# B&R Automation Studio project BR_ZBM1
Automation Studio 4.1.5.68 SP

## Configuration Config1

CPU , AutomationRuntime K4.06, Build 4.1.2

### Task classes (Cpu.sw)
```
Cyclic#4 (cycle 100000 us, tolerance 100000 us):
  BU_2 <- BunchUnits.BU_2.prg
  can_diag <- Exceptionhandling.can_diag.prg
  SC_2 <- BunchUnits.SC_2.prg
VcDataObjects: Mobile <- Visualisation.Mobile.dob
Binaries: asfw, ashwd, arconfig, sysconf, iomap
Libraries: standard, astime, runtime, asieccon, Hardware
```

### Hardware
```
X20CP1586 : X20CP1586 v1.0.5.0
  Connector IF2:
    ActivateDevice = 1
    Mode = Manual
    InternetAddress = 192.168.0.1
    SubnetMask = 255.255.255.0
  Cyclic1Duration = 1000
  Cyclic1Tolerance = 10000
  Cyclic2Duration = 20000
  Cyclic2Tolerance = 20000
  Cyclic3Duration = 50000
  Cyclic3Tolerance = 50000
  Cyclic4Duration = 100000
  Cyclic4Tolerance = 100000
  Cyclic5Duration = 200000
  Cyclic5Tolerance = 200000
  Cyclic6Duration = 500000
  Cyclic6Tolerance = 500000
  Cyclic7Duration = 1000000
  Cyclic7Tolerance = 1000000
  Cyclic8Duration = 10000
  Cyclic8Tolerance = 30000000
```

### IoMap.iom - X20CP1586/IoMap.iom
```iecst
(********************************************************************
 * COPYRIGHT -- Bernecker + Rainer
 ********************************************************************
 * File: IoMap.iom
 * Author: frankenj
 * Created: December 04, 2014
 ********************************************************************
 * IO mapping file
 ********************************************************************)
VAR_CONFIG
	::myPulseUse:linkedSystemTime AT %ID."X20CP1586".SystemTime;
END_VAR
```

## Configuration X20

CPU X20CP1585, AutomationRuntime C4.09, Build 4.1.2

### Task classes (Cpu.sw)
```
Cyclic#1 (cycle 1000 us, tolerance 0 us):
  Shiftregis <- MainControlUnit.Shiftregister.prg  // Control for chain sensor
  Simulation <- MainControlUnit.Simulation.prg
  Main <- MainControlUnit.Main.prg
Cyclic#2 (cycle 5000 us, tolerance 0 us):
  IOpolling <- IOHandling.IOpolling.prg
  BeltContro <- MainBeltUnit.BeltControl.prg
Cyclic#3 (cycle 50000 us, tolerance 0 us):
  RS_I <- BunchUnits.RS_I.prg
  BU_1 <- BunchUnits.BU_1.prg
  SC_1 <- BunchUnits.SC_1.prg
  BU_2 <- BunchUnits.BU_2.prg
  SC_2 <- BunchUnits.SC_2.prg
  BU_3 <- BunchUnits.BU_3.prg
  SC_3 <- BunchUnits.SC_3.prg
  BU_4 <- BunchUnits.BU_4.prg
  SC_4 <- BunchUnits.SC_4.prg
  BU_5 <- BunchUnits.BU_5.prg
  SC_5 <- BunchUnits.SC_5.prg
  BU_6 <- BunchUnits.BU_6.prg
  SC_6 <- BunchUnits.SC_6.prg
  BU_7 <- BunchUnits.BU_7.prg
  SC_7 <- BunchUnits.SC_7.prg
  BU_8 <- BunchUnits.BU_8.prg
  SC_8 <- BunchUnits.SC_8.prg
  BU_9 <- BunchUnits.BU_9.prg
  SC_9 <- BunchUnits.SC_9.prg
  BU_10 <- BunchUnits.BU_10.prg
  SC_10 <- BunchUnits.SC_10.prg
Cyclic#4 (cycle 100000 us, tolerance 0 us):
  ErrorHandl <- Exceptionhandling.ErrorHandling.prg
  can_diag <- Exceptionhandling.can_diag.prg
Cyclic#5 (cycle 10000 us, tolerance 30000000 us):
  Init <- BunchUnits.Init.prg
  Sender <- Lichtkrant.Sender.prg
VcDataObjects: BU_Gui <- Visualisation.BU_Gui_Resized.dob [disabled], Mobile <- Visualisation.Mobile.dob [disabled]
Binaries: OpcUaMap, sysconf, iomap, ashwd, asfw, arconfig, asnxdb2, vcchspot, asnxdb1, vccbar, vcclbox, vcchtml, vccstr, vccline, vccscale, vccalarm, vccgauge, vccurl, vcxml, vcpfar00, vccnum, arialbd, vcdsloc, vcfntttf, vcdsint, vcshared, vcrt, vcbclass, vcfile, vccbtn, vcresman, vcalarm, vcpdsw, arial, vccovl, vcgclass, Mobile02, Mobile03, vccddbox, vccpopup, vccdt, vcctext, vccshape, vccbmp, vcctrend, BU_Gui02, BU_Gui03, vccslider, vcmgr, vcnet, vcpkat, vctcal, BU_Gui01, vcpdvnc, vcpfx20, Mobile01
Libraries: sys_lib, Runtime, astime, asieccon, AsTCP, brsystem, asstring, standard, PulsGen, AsNxCoM, Inverter, BULib, Servo, SDO, dvframe, Lichtkrant, Chain, AsBrStr, hex2dec, Serial, SensContr, MBU_lib, IecCheck, AsArLog, Hardware, dataobj, fileio, ashw
```

### Hardware
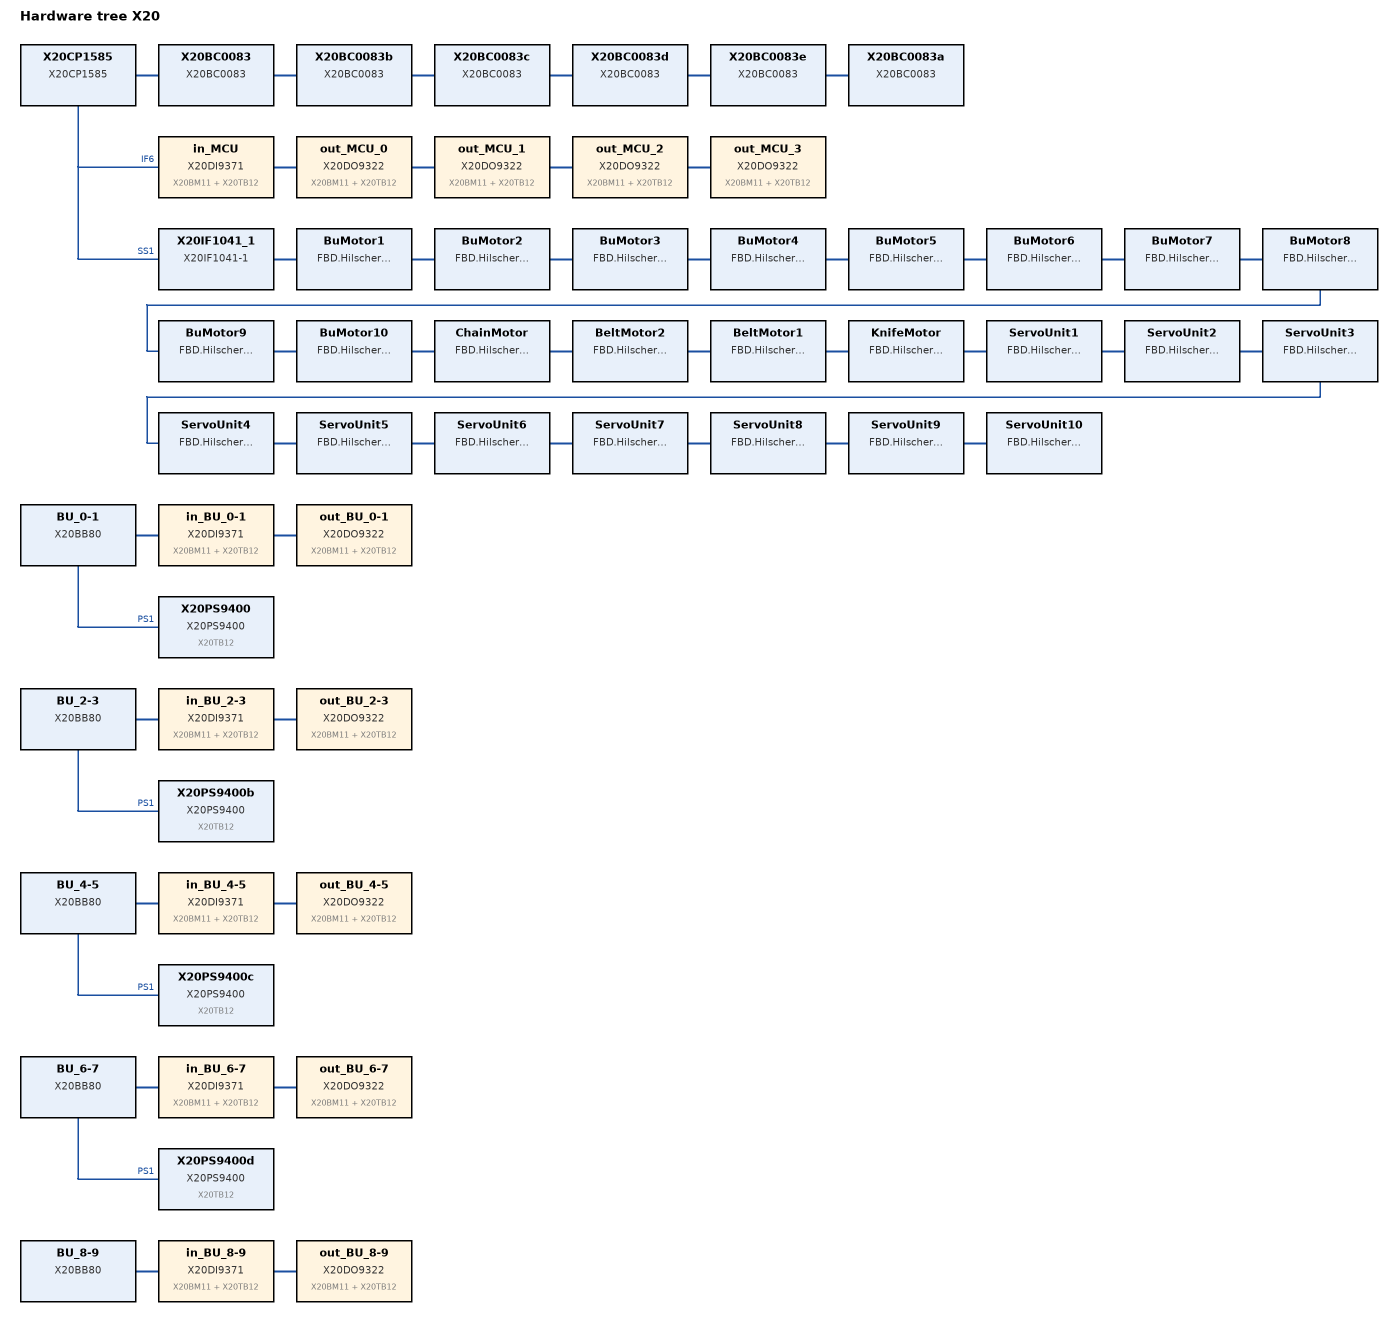
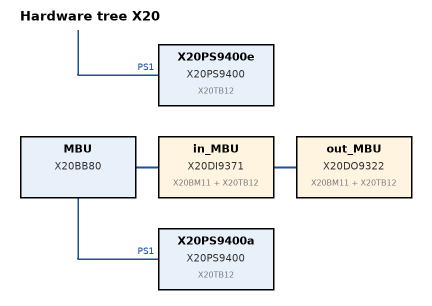
```
BeltMotor1 : FBD.Hilscher.COGenSlaveDTM.ACOPOSinverter X64 (ACOPOSinverter_X64.eds) v0.0.0.0 (OrderNumber=ACOPOSinverter_X64__ACOPOSinverter_X64_eds_)  [CAN1 -> BeltMotor2.CAN2 (NodeNumber=4)]
  DtmId = 0e41fe58-9b29-4e80-aa17-b3b9a602be41
  ChannelBlocks_54c748ae-a862-45bf-bd05-307df38cf45a  // Receive PDO1 parameter
  IO_aca35ca7-9daa-4f2c-a263-cb1312a79025  // 2 Byte(s)
  ChannelBlocks_6fc9c6dd-ef6a-4241-a49b-47093041261e  // Receive PDO6 parameter
  IO_a09422e8-9296-4dde-995f-c21dba077c83  // 2 Byte(s)
  IO_c6b60006-1097-4b2b-99a2-873ae92355e9  // 2 Byte(s)
  IO_be17ac07-0c86-4ed7-8a83-77242752eabc  // 2 Byte(s)
  ChannelBlocks_0de3404d-a2ba-475d-9759-ce1c75ca456f  // Transmit PDO1 parameter
  IO_d4d6ac5b-6312-46c0-bea3-1feb3fe2ff1b  // 2 Byte(s)
  ChannelBlocks_35f5ad43-0655-49b5-a722-94d15f201f4c  // Transmit PDO6 parameter
  IO_54646803-abb9-4e9d-b295-57a01534b6c3  // 2 Byte(s)
  IO_ae920d2b-a2b1-4de3-a1c4-e574386f93fb  // 2 Byte(s)
  IO_47f71d08-67d5-4a29-b608-1e0426a373c3  // 2 Byte(s)
  IO_76edcae2-a5b3-42ff-aea4-90ff8a7df386  // 2 Byte(s)
BeltMotor2 : FBD.Hilscher.COGenSlaveDTM.ACOPOSinverter X64 (ACOPOSinverter_X64.eds) v0.0.0.0 (OrderNumber=ACOPOSinverter_X64__ACOPOSinverter_X64_eds_)  [CAN1 -> ChainMotor.CAN2 (NodeNumber=5)]
  DtmId = 5224c894-1ef8-4fa5-9f2e-7023e8237f50
  ChannelBlocks_54ef21bf-51ac-4b79-9d7d-aaf36440fde1  // Receive PDO1 parameter
  IO_08901fce-ce4a-45a7-8fa1-4352fddaeca0  // 2 Byte(s)
  ChannelBlocks_5fdfdc2d-6504-40c7-b6e9-5c26043bbabb  // Receive PDO6 parameter
  IO_7efb87b6-7525-4814-82a4-a00de786267e  // 2 Byte(s)
  IO_1c5a6fdf-985c-41b4-867c-db4a3086964a  // 2 Byte(s)
  IO_89f973fb-223e-4f5d-b0cf-d7557db3c308  // 2 Byte(s)
  ChannelBlocks_ff6de664-0730-4c0c-a004-c59824083d59  // Transmit PDO1 parameter
  IO_6a6c6cea-e364-4156-9bd8-734b31d4d8b2  // 2 Byte(s)
  ChannelBlocks_b2f2cbd0-76eb-4694-9316-88ecd34e890c  // Transmit PDO6 parameter
  IO_27630f78-04b9-4817-a004-ac8ed4a34943  // 2 Byte(s)
  IO_a532a8b0-ae79-4199-8f10-aceb97e86d8c  // 2 Byte(s)
  IO_80c1adba-b4c6-4671-a8d4-c5debac3ab04  // 2 Byte(s)
  IO_db551fcc-40d8-4d75-964b-d0c34238111c  // 2 Byte(s)
BU_0-1 : X20BB80 v1.0.0.2
  Connector IF1:
    BusLength = 100
BU_2-3 : X20BB80 v1.0.0.2
BU_4-5 : X20BB80 v1.0.0.2
BU_6-7 : X20BB80 v1.0.0.2
BU_8-9 : X20BB80 v1.0.0.2
BuMotor1 : FBD.Hilscher.COGenSlaveDTM.ACOPOSinverter X64 (ACOPOSinverter_X64.eds) v0.0.0.0 (OrderNumber=ACOPOSinverter_X64__ACOPOSinverter_X64_eds_)  [CAN1 -> X20IF1041_1.IF1 (NodeNumber=10)]
  DtmId = 41eacdba-3555-4f40-ac61-2c8428ea58b2
  ChannelBlocks_b9ddc844-9481-4af5-a747-25b3e2109658  // Receive PDO1 parameter
  IO_7b4bc88c-5ce5-4aaa-a58d-90f33b48a65c  // 2 Byte(s)
  ChannelBlocks_8b5f3c6e-1732-4951-a210-c4de25588974  // Receive PDO6 parameter
  IO_39a2cd53-b850-4b06-8776-b6d11eb43720  // 2 Byte(s)
  IO_30629477-0436-4440-ba53-af916bfbef45  // 2 Byte(s)
  IO_eda63b9e-3d56-4a36-8c45-b6b1969d639a  // 2 Byte(s)
  ChannelBlocks_f1365d26-9917-401f-a453-e6262fccb88e  // Transmit PDO1 parameter
  IO_8b996910-5de3-45a7-9e18-c98469aeffd6  // 2 Byte(s)
  ChannelBlocks_48485091-4447-4b08-b8f7-2a8039d8dcd2  // Transmit PDO6 parameter
  IO_be2a3e1f-8d08-4dea-a2d2-a29b4de4c830  // 2 Byte(s)
  IO_55fef0e3-e778-4333-8784-725b71533f49  // 2 Byte(s)
  IO_626eea93-30a0-479c-9321-2dd4622e8684  // 2 Byte(s)
  IO_53a93a48-f76d-4478-8b66-bfaf7ee8cb03  // 2 Byte(s)
BuMotor10 : FBD.Hilscher.COGenSlaveDTM.ACOPOSinverter X64 (ACOPOSinverter_X64.eds) v0.0.0.0 (OrderNumber=ACOPOSinverter_X64__ACOPOSinverter_X64_eds_)  [CAN1 -> BuMotor9.CAN2 (NodeNumber=28)]
  DtmId = 334ec416-5c16-4925-9ab1-88c2f19d51fb
  ChannelBlocks_ac9c813b-77a1-48ff-9722-79a7e36309a3  // Receive PDO1 parameter
  IO_4aa75d45-937a-4143-8e5e-5239ec3df5d5  // 2 Byte(s)
  ChannelBlocks_bd99a9ef-60c2-4465-b2ca-5589d312d023  // Receive PDO6 parameter
  IO_10874e3a-ea7a-435e-b16d-3cfd83cd96d2  // 2 Byte(s)
  IO_a0da98ff-73a6-482d-a789-9eea3a9ef5ec  // 2 Byte(s)
  IO_a035e9e4-fedc-44f8-8d04-fa4482e8e6f6  // 2 Byte(s)
  ChannelBlocks_c4ede1fb-b8c3-46bc-aa40-d6c07d995dd8  // Transmit PDO1 parameter
  IO_3a67936d-7775-49f5-8896-9a8e4e400f8a  // 2 Byte(s)
  ChannelBlocks_4cda3d3d-ce84-47df-a9c8-383005e5aed1  // Transmit PDO6 parameter
  IO_f52c2df5-83ca-4265-9fb6-a04d781d80b2  // 2 Byte(s)
  IO_496498d8-ae6d-4630-839d-faafd4532c16  // 2 Byte(s)
  IO_a3e387be-6efa-4130-b18c-b95da0514b42  // 2 Byte(s)
  IO_b0e32a9b-b548-480f-ab2f-b0d362bbdba9  // 2 Byte(s)
BuMotor2 : FBD.Hilscher.COGenSlaveDTM.ACOPOSinverter X64 (ACOPOSinverter_X64.eds) v0.0.0.0 (OrderNumber=ACOPOSinverter_X64__ACOPOSinverter_X64_eds_)  [CAN1 -> BuMotor1.CAN2 (NodeNumber=12)]
  DtmId = e1ce438d-8ff1-4ad6-81a8-1a105d1b79ee
  ChannelBlocks_303446a4-05f8-4f0b-b2b4-7c1333c2b877  // Receive PDO1 parameter
  IO_edbfdedc-cf52-4617-8a63-87053fac3909  // 2 Byte(s)
  ChannelBlocks_72fe8bc7-9e89-4c3c-9af8-bb7ce4d6a99e  // Receive PDO6 parameter
  IO_7fc3c5cf-f8f6-4322-9a74-de616acc70eb  // 2 Byte(s)
  IO_f67c0509-47e2-4490-9eac-614590cde9d6  // 2 Byte(s)
  IO_987d5f71-5d59-414d-b133-eb996a41fb68  // 2 Byte(s)
  ChannelBlocks_1b47f333-0257-4114-959e-33d260186bf4  // Transmit PDO1 parameter
  IO_6f79accf-2d80-4323-98c0-77cea77bfb60  // 2 Byte(s)
  ChannelBlocks_efe37a9e-d3f3-48e1-a345-23b1c1da338c  // Transmit PDO6 parameter
  IO_a5a00cb8-1081-40a9-aa27-5251b345f7d4  // 2 Byte(s)
  IO_3161684f-0b69-4f3b-957e-df44177686f9  // 2 Byte(s)
  IO_430b3064-68ec-4c3e-8c05-6340c25ce5c7  // 2 Byte(s)
  IO_47871665-a16d-49f5-80b8-ccf6bf5cb8a7  // 2 Byte(s)
BuMotor3 : FBD.Hilscher.COGenSlaveDTM.ACOPOSinverter X64 (ACOPOSinverter_X64.eds) v0.0.0.0 (OrderNumber=ACOPOSinverter_X64__ACOPOSinverter_X64_eds_)  [CAN1 -> BuMotor2.CAN2 (NodeNumber=14)]
  DtmId = 1e61ad36-4c2a-4e56-bdd1-0d91381fff01
  ChannelBlocks_16131e21-e2ce-44a8-8d6c-ee170c9dd84c  // Receive PDO1 parameter
  IO_233081b4-53a4-47f1-884f-f2efd1a08929  // 2 Byte(s)
  ChannelBlocks_53a3e1b0-6088-4904-962c-d97f114e68db  // Receive PDO6 parameter
  IO_e6106a2d-9b03-4786-b4da-5020b8cc5489  // 2 Byte(s)
  IO_0f48f256-f7be-491a-8248-9956108b6aa0  // 2 Byte(s)
  IO_afc01347-6de2-439e-b259-33123674c101  // 2 Byte(s)
  ChannelBlocks_5db5365c-7f68-4bfd-af2b-a09bb430efe1  // Transmit PDO1 parameter
  IO_cfab9ccf-d03f-406c-96ae-dbf087d83766  // 2 Byte(s)
  ChannelBlocks_e96627b7-b6f5-430a-82cb-a06f050c10a1  // Transmit PDO6 parameter
  IO_7d74f071-110e-4899-967d-10e546879826  // 2 Byte(s)
  IO_ff055412-aa6d-43cc-975d-a3aff2303c44  // 2 Byte(s)
  IO_c96c42f2-eb3c-407f-abc8-e2aec00ccd6f  // 2 Byte(s)
  IO_9c4becff-3ca0-4837-b00f-01cea90c8b43  // 2 Byte(s)
BuMotor4 : FBD.Hilscher.COGenSlaveDTM.ACOPOSinverter X64 (ACOPOSinverter_X64.eds) v0.0.0.0 (OrderNumber=ACOPOSinverter_X64__ACOPOSinverter_X64_eds_)  [CAN1 -> BuMotor3.CAN2 (NodeNumber=16)]
  DtmId = 3419c233-701d-4c2b-a99c-e2e251ebd402
  ChannelBlocks_e8b2e42e-dc9f-4e9b-afe3-218e25b141be  // Receive PDO1 parameter
  IO_16dab77e-f7aa-424b-acc6-a2f3740772d1  // 2 Byte(s)
  ChannelBlocks_3a5654fc-b013-413b-88ca-ad42da5e8159  // Receive PDO6 parameter
  IO_0fc3cbd3-a556-4aa9-b6b1-565b33da217c  // 2 Byte(s)
  IO_f37a6bc4-d7ce-4ecd-85ac-62dd2e5de9aa  // 2 Byte(s)
  IO_04a94dea-b5f7-4965-bf5b-fca15ddf3456  // 2 Byte(s)
  ChannelBlocks_fb4caf4b-a8c9-44e0-a0df-9b1c4a38039a  // Transmit PDO1 parameter
  IO_32d90893-e468-4b93-b87b-e735c85ecb31  // 2 Byte(s)
  ChannelBlocks_84a463cb-60ca-4f79-80bc-efdcbf518684  // Transmit PDO6 parameter
  IO_af34fa9f-553d-4e33-8a4e-a96a9d17e081  // 2 Byte(s)
  IO_52b55ddc-0196-4b87-8ece-0689d53c35ee  // 2 Byte(s)
  IO_ece82347-fffd-4285-b914-98d6765bff2c  // 2 Byte(s)
  IO_ecb960f2-7d71-49be-b58a-71f34bd8c015  // 2 Byte(s)
BuMotor5 : FBD.Hilscher.COGenSlaveDTM.ACOPOSinverter X64 (ACOPOSinverter_X64.eds) v0.0.0.0 (OrderNumber=ACOPOSinverter_X64__ACOPOSinverter_X64_eds_)  [CAN1 -> BuMotor4.CAN2 (NodeNumber=18)]
  DtmId = 4c32e5ad-4edb-4bc3-84fb-2c963843a420
  ChannelBlocks_3b0e43e7-5611-43d6-8ec6-2ede2cec3a32  // Receive PDO1 parameter
  IO_bb960a29-c17d-45e9-ae40-da831eee433e  // 2 Byte(s)
  ChannelBlocks_9aa1925c-833d-4633-8e49-89084995cc3b  // Receive PDO6 parameter
  IO_a9c7e03e-2a47-4cfa-95a2-7cf40ba5363c  // 2 Byte(s)
  IO_55832d8a-1481-4b90-82e1-34e4fb78b3e2  // 2 Byte(s)
  IO_e57ca11a-3f47-4da8-8504-ed0e9a8a8339  // 2 Byte(s)
  ChannelBlocks_132f04aa-a5a6-49b1-b157-8f99cfa41fb9  // Transmit PDO1 parameter
  IO_d17d2007-b5bc-4df8-874a-5af49acdc510  // 2 Byte(s)
  ChannelBlocks_cb051f0a-81b6-44f0-a47a-0639dce175ec  // Transmit PDO6 parameter
  IO_0ab8f150-63b8-41c9-817d-7015de8b9c0b  // 2 Byte(s)
  IO_fee015dc-7fc2-42a9-8830-1e4733cc798a  // 2 Byte(s)
  IO_6cbc9beb-0f89-432a-b861-7296453a7b1e  // 2 Byte(s)
  IO_2e4c1757-1ae4-40e8-a121-0788d8ac6cc6  // 2 Byte(s)
BuMotor6 : FBD.Hilscher.COGenSlaveDTM.ACOPOSinverter X64 (ACOPOSinverter_X64.eds) v0.0.0.0 (OrderNumber=ACOPOSinverter_X64__ACOPOSinverter_X64_eds_)  [CAN1 -> BuMotor5.CAN2 (NodeNumber=20)]
  DtmId = 212c5dca-78b8-435a-aa98-aeeae71d2177
  ChannelBlocks_36548871-ea81-46d0-ab51-c23f60eb9c43  // Receive PDO1 parameter
  IO_972244c1-2427-47a5-b961-02e0ea3bca84  // 2 Byte(s)
  ChannelBlocks_8e6d6cc0-2f64-493a-b846-8f9fde6f0b95  // Receive PDO6 parameter
  IO_43c1df8f-fc75-4873-b39e-321cf2aeae78  // 2 Byte(s)
  IO_93ac0147-b909-4f64-8bd2-362413b76dca  // 2 Byte(s)
  IO_6dd5a1a6-fcdb-48f0-a691-0d50ab35e40a  // 2 Byte(s)
  ChannelBlocks_b0830481-7508-4cb8-bd75-74145b1e5a65  // Transmit PDO1 parameter
  IO_78f69379-eb6e-4920-aad6-d2f1523e5569  // 2 Byte(s)
  ChannelBlocks_d19e3ad9-8e69-4d25-8d92-be2b259d078d  // Transmit PDO6 parameter
  IO_df6299ac-0345-46ea-9f36-596b15d796e2  // 2 Byte(s)
  IO_93665609-78bd-4ea5-b921-8d6c30ac71e7  // 2 Byte(s)
  IO_692a70c6-2a2e-4ad9-904d-ad6ece7e714a  // 2 Byte(s)
  IO_0b12c3e3-a068-4783-a61b-308601e6b628  // 2 Byte(s)
BuMotor7 : FBD.Hilscher.COGenSlaveDTM.ACOPOSinverter X64 (ACOPOSinverter_X64.eds) v0.0.0.0 (OrderNumber=ACOPOSinverter_X64__ACOPOSinverter_X64_eds_)  [CAN1 -> BuMotor6.CAN2 (NodeNumber=22)]
  DtmId = fe6d1ec7-057d-4e3d-8429-4d9d0807c15d
  ChannelBlocks_23640bc2-8a9b-4e0c-99a5-9585fc2825da  // Receive PDO1 parameter
  IO_c5a90a3b-2ea9-45c8-8169-e1e808272f75  // 2 Byte(s)
  ChannelBlocks_7172327e-45a5-44f5-ad87-af72047464ff  // Receive PDO6 parameter
  IO_f30a1fbe-7a72-4da2-8571-4465ed769e94  // 2 Byte(s)
  IO_3bb66d1e-0ded-48ae-8f3a-aaeca947f466  // 2 Byte(s)
  IO_05489d67-538a-494e-9c37-4f3ed3ae3460  // 2 Byte(s)
  ChannelBlocks_7646f274-a7ae-4c51-9912-41f9c3be717f  // Transmit PDO1 parameter
  IO_b8501f12-b2ac-4cca-aa30-82df59980588  // 2 Byte(s)
  ChannelBlocks_60981db9-e146-4d25-8f47-02ae1f72b5ae  // Transmit PDO6 parameter
  IO_9564daf5-683d-42b1-a2ba-dbdcc986d03e  // 2 Byte(s)
  IO_1d121221-d496-428f-9b5b-e106d2b53480  // 2 Byte(s)
  IO_132e6c0a-0438-441f-a77f-0b8e58432b79  // 2 Byte(s)
  IO_fed1b959-84a4-4ae2-be07-728b9434a0fb  // 2 Byte(s)
BuMotor8 : FBD.Hilscher.COGenSlaveDTM.ACOPOSinverter X64 (ACOPOSinverter_X64.eds) v0.0.0.0 (OrderNumber=ACOPOSinverter_X64__ACOPOSinverter_X64_eds_)  [CAN1 -> BuMotor7.CAN2 (NodeNumber=24)]
  DtmId = d0e7570d-e994-4edf-9e81-ec8efb494bdc
  ChannelBlocks_1c234084-f26d-4010-ae60-430dc9ea6039  // Receive PDO1 parameter
  IO_f51d2d11-2100-42d4-9367-ddf86f21ba8a  // 2 Byte(s)
  ChannelBlocks_bc9900bd-4277-4d30-ab2b-fc45edb7799e  // Receive PDO6 parameter
  IO_e6a06380-dc77-42c1-8abc-946aceaaeec3  // 2 Byte(s)
  IO_b998704f-b9a3-4a2e-a70b-97f25279deec  // 2 Byte(s)
  IO_27fd5a55-6180-49bd-8ed4-b0dfe1ebd659  // 2 Byte(s)
  ChannelBlocks_ad54a2c5-da08-4f7b-a056-b92f63750228  // Transmit PDO1 parameter
  IO_ac97c997-ad95-465a-b815-b5fc32ccf499  // 2 Byte(s)
  ChannelBlocks_6dc4ac7d-db58-431d-9a69-65407098d216  // Transmit PDO6 parameter
  IO_621d38ea-a82c-463b-832d-9b3839800169  // 2 Byte(s)
  IO_0795fb83-6342-4703-bf59-004121218c89  // 2 Byte(s)
  IO_4a80c6ec-6f72-4231-92da-efd4b17a3a1c  // 2 Byte(s)
  IO_8daf75e9-a6d5-4c91-9108-ab4f8b4fc76f  // 2 Byte(s)
BuMotor9 : FBD.Hilscher.COGenSlaveDTM.ACOPOSinverter X64 (ACOPOSinverter_X64.eds) v0.0.0.0 (OrderNumber=ACOPOSinverter_X64__ACOPOSinverter_X64_eds_)  [CAN1 -> BuMotor8.CAN2 (NodeNumber=26)]
  DtmId = 27a4961f-41ec-4434-a3f4-61cbc6fb7192
  ChannelBlocks_156d82cd-4cce-4b22-929c-902f2fb9b58d  // Receive PDO1 parameter
  IO_8583cb26-f389-4261-951d-3ac93a53ae0b  // 2 Byte(s)
  ChannelBlocks_af10b2dc-1205-4d97-96ea-c7d2b9fb63c2  // Receive PDO6 parameter
  IO_e5a889ae-0a76-469a-b754-943b3c45a784  // 2 Byte(s)
  IO_43edfdd7-2d01-4208-a7b9-dc719fad88a4  // 2 Byte(s)
  IO_8c64ee22-0973-473c-b1a9-8b58114fd87f  // 2 Byte(s)
  ChannelBlocks_7bc1f4a0-5bf3-43fa-882a-01fc853e14d7  // Transmit PDO1 parameter
  IO_3c1e0984-52c5-4e10-9971-b2afe92d426d  // 2 Byte(s)
  ChannelBlocks_a95ce928-01d1-410a-a36f-9f939e55dbb5  // Transmit PDO6 parameter
  IO_83dbfe57-663e-4119-9086-e5341eb48c58  // 2 Byte(s)
  IO_dd747ed3-faa4-4833-823f-d91767ba62f9  // 2 Byte(s)
  IO_ff04d007-1200-431c-b421-f6f4c823914d  // 2 Byte(s)
  IO_53450f9b-88e3-4ab2-bf5f-c81ceddf348f  // 2 Byte(s)
ChainMotor : FBD.Hilscher.COGenSlaveDTM.ACOPOSinverter X64 (ACOPOSinverter_X64.eds) v0.0.0.0 (OrderNumber=ACOPOSinverter_X64__ACOPOSinverter_X64_eds_)  [CAN1 -> BuMotor10.CAN2 (NodeNumber=2)]
  DtmId = a1bf2b9b-c770-4510-aeb7-956fae696789
  ChannelBlocks_ab51fc66-ccfe-4969-aa09-56bf748c4a12  // Receive PDO1 parameter
  IO_db442f5f-1e91-4533-b5dd-19ba2275383e  // 2 Byte(s)
  ChannelBlocks_ae38ce3c-268a-4902-ab02-c82d525d9cbb  // Receive PDO6 parameter
  IO_ecf49792-71fd-4e43-b62d-26aec71b8eab  // 2 Byte(s)
  IO_62c798e0-2415-4177-bd7c-f597b6d9ce16  // 2 Byte(s)
  IO_d3603888-cc95-456b-b613-e3c0c1640d24  // 2 Byte(s)
  ChannelBlocks_115e84f3-a25d-449a-a537-95b5558b7c26  // Transmit PDO1 parameter
  IO_9748ba3b-e319-4fcf-8e43-a2aead93d9d4  // 2 Byte(s)
  ChannelBlocks_95271bd8-90e8-4465-a473-25a5ce2b8c1d  // Transmit PDO6 parameter
  IO_3683007d-d99b-4002-825a-f0003ae249a9  // 2 Byte(s)
  IO_d93fc321-8f8b-45f1-8332-7d1270e96476  // 2 Byte(s)
  IO_8b5f3a95-c21d-40c8-ae74-161c5e85b92d  // 2 Byte(s)
  IO_57e4cc6a-288c-4cc7-b99a-80fc403e645e  // 2 Byte(s)
in_BU_0-1 : X20DI9371 v1.0.1.2  [SS1 -> X20TB12.SS; SL -> X20BM11.SL1]
  Supervision = off
in_BU_2-3 : X20DI9371 v1.0.1.2  [SS1 -> X20TB12o.SS; SL -> X20BM11i.SL1]
  Supervision = off
in_BU_4-5 : X20DI9371 v1.0.1.2  [SS1 -> X20TB12p.SS; SL -> X20BM11j.SL1]
  Supervision = off
in_BU_6-7 : X20DI9371 v1.0.1.2  [SS1 -> X20TB12q.SS; SL -> X20BM11k.SL1]
  Supervision = off
in_BU_8-9 : X20DI9371 v1.0.1.2  [SS1 -> X20TB12r.SS; SL -> X20BM11l.SL1]
  Supervision = off
in_MBU : X20DI9371 v1.0.1.2  [SS1 -> X20TB12i.SS; SL -> X20BM11g.SL1]
  Supervision = off
in_MCU : X20DI9371 v1.0.1.2  [SS1 -> X20TB12g.SS; SL -> X20BM11f.SL1]
  Supervision = off
  InputFilter = 1
KnifeMotor : FBD.Hilscher.COGenSlaveDTM.ACOPOSinverter X64 (ACOPOSinverter_X64.eds) v0.0.0.0 (OrderNumber=ACOPOSinverter_X64__ACOPOSinverter_X64_eds_)  [CAN1 -> BeltMotor1.CAN2 (NodeNumber=6)]
  DtmId = 33a85843-c74d-4b86-b247-01135a679646
  ChannelBlocks_959f5f2a-c98d-43ac-ab77-7afc3a4601f4  // Receive PDO1 parameter
  IO_518f3516-227d-4baa-b2e9-9837cdbd9b05  // 2 Byte(s)
  ChannelBlocks_e5b71d72-a2cb-487c-afa4-c76067c8cb50  // Receive PDO6 parameter
  IO_fae67bf3-6369-40bc-b0b3-d34df1ae89ca  // 2 Byte(s)
  IO_6eee8b06-f52d-4686-a1ea-7920ca6ed831  // 2 Byte(s)
  IO_f2afe01e-1957-4460-af08-4c926f12efa2  // 2 Byte(s)
  ChannelBlocks_fb08993c-509f-478c-8a17-eacbe3bef14b  // Transmit PDO1 parameter
  IO_42e58779-80ce-41f3-942d-bae492baa4fc  // 2 Byte(s)
  ChannelBlocks_d914b564-1111-4bb5-90f7-738445a3305b  // Transmit PDO6 parameter
  IO_dc6d6c3f-094b-44a2-a37e-299af11b9a90  // 2 Byte(s)
  IO_82bcc08e-10b1-46a3-8141-af866fd3a5d5  // 2 Byte(s)
  IO_10a6ed0e-5e2a-46a1-9302-e179eca58b81  // 2 Byte(s)
  IO_25f6a930-9e41-48f9-ae4a-248184c6394c  // 2 Byte(s)
MBU : X20BB80 v1.0.0.2
out_BU_0-1 : X20DO9322 v1.0.2.2  [SS1 -> X20TB12c.SS; SL -> X20BM11b.SL1]
  Supervision = off
out_BU_2-3 : X20DO9322 v1.0.2.2  [SS1 -> X20TB12s.SS; SL -> X20BM11m.SL1]
  Supervision = off
out_BU_4-5 : X20DO9322 v1.0.2.2  [SS1 -> X20TB12t.SS; SL -> X20BM11n.SL1]
  Supervision = off
out_BU_6-7 : X20DO9322 v1.0.2.2  [SS1 -> X20TB12u.SS; SL -> X20BM11o.SL1]
  Supervision = off
out_BU_8-9 : X20DO9322 v1.0.2.2  [SS1 -> X20TB12v.SS; SL -> X20BM11p.SL1]
  Supervision = off
out_MBU : X20DO9322 v1.0.2.2  [SS1 -> X20TB12j.SS; SL -> X20BM11h.SL1]
  Supervision = off
out_MCU_0 : X20DO9322 v1.0.2.2  [SS1 -> X20TB12b.SS; SL -> X20BM11a.SL1]
  Supervision = off
out_MCU_1 : X20DO9322 v1.0.2.2  [SS1 -> X20TB12d.SS; SL -> X20BM11c.SL1]
  Supervision = off
out_MCU_2 : X20DO9322 v1.0.2.2  [SS1 -> X20TB12f.SS; SL -> X20BM11e.SL1]
  Supervision = off
out_MCU_3 : X20DO9322 v1.0.2.2  [SS1 -> X20TB12e.SS; SL -> X20BM11d.SL1]
  Supervision = off
ServoUnit1 : FBD.Hilscher.COGenSlaveDTM.CMMS-ST (FHPP) (CMMS-ST_CAN_FHPP.eds) v0.0.0.0 (OrderNumber=CMMS_ST__FHPP___CMMS_ST_CAN_FHPP_eds_)  [CAN1 -> KnifeMotor.CAN2 (NodeNumber=11)]
  DtmId = 2cc01d8c-52a8-4f03-b874-cf26b4fa5fc9
  ChannelBlocks_f65e5b16-ad22-40ee-992f-65e9134c0818  // receive_pdo_parameter_RPDO1
  IO_7413fdc9-d251-41aa-a295-413caee91bb0  // 1 Byte(s)
  IO_8c39c384-d077-4c2a-ac09-6e48e9cd8298  // 1 Byte(s)
  IO_5b4e01b4-bc10-43d6-990c-ca8cf807684f  // 1 Byte(s)
  IO_2912853e-21ed-466d-b4af-a4ce6ec0f99a  // 1 Byte(s)
  IO_54c5027d-38d4-4e0c-80b9-518f4f6d60ce  // 4 Byte(s)
  ChannelBlocks_3cd1045e-a7fe-4c41-b716-5963c2d0f415  // receive_pdo_parameter_RPDO2
  IO_02894f07-1dcd-4eb4-970d-ac259e8bc589  // 1 Byte(s)
  IO_1110f2e0-e843-4e28-bbeb-fa5d8a28fd9b  // 1 Byte(s)
  IO_5de8c302-b593-409f-a351-0f865c6bfcd2  // 2 Byte(s)
  IO_f43418fd-0be3-49b4-9f0a-46c06fad4ee0  // 4 Byte(s)
  ChannelBlocks_69007e23-4ad5-47fe-8b89-c8cf6e8d2953  // transmit_pdo_parameter_TPDO1
  IO_02be1259-9179-42ca-a2b1-1ec2453c51ec  // 1 Byte(s)
  IO_f7942894-44d6-4bab-941f-fefb330485f5  // 1 Byte(s)
  IO_ffab8801-ccee-4f54-afc8-b18e81cc8d53  // 1 Byte(s)
  IO_230f5946-6524-4ad5-9596-a8270efa9ae4  // 1 Byte(s)
  IO_5e14c759-19f2-47bd-845a-76715e6b65ec  // 4 Byte(s)
  ChannelBlocks_ac1dc8db-3e8f-49dc-9bd9-dac3f25cea3b  // transmit_pdo_parameter_TPDO2
  IO_50fa45dc-06c8-4e45-86a5-632600e82df9  // 1 Byte(s)
  IO_dcaa8277-d514-4b77-8c9c-59ea68ad03d1  // 1 Byte(s)
  IO_2b895b55-3353-4bb0-9d55-88662917902a  // 2 Byte(s)
  IO_96caa5a3-b367-4c2d-91d3-4c9d541150a0  // 4 Byte(s)
ServoUnit10 : FBD.Hilscher.COGenSlaveDTM.CMMS-ST (FHPP) (CMMS-ST_CAN_FHPP.eds) v0.0.0.0 (OrderNumber=CMMS_ST__FHPP___CMMS_ST_CAN_FHPP_eds_)  [CAN1 -> ServoUnit9.CAN2 (NodeNumber=29)]
  DtmId = a13dd3ca-1f37-4c54-a947-4a4feb01707b
  ChannelBlocks_91fa1f26-9aaa-436b-b26e-7c56dcb6ef4f  // receive_pdo_parameter_RPDO1
  IO_15dbd178-5c5a-43b8-b447-b7434bae5630  // 1 Byte(s)
  IO_77cb988d-107f-444c-9931-909d67709d08  // 1 Byte(s)
  IO_d28c5ade-4123-4660-a144-0029614273c4  // 1 Byte(s)
  IO_f58dc55c-0554-491a-9586-ae74ffbb8fc9  // 1 Byte(s)
  IO_026e0246-a0ce-4501-8433-2dbe8596be8f  // 4 Byte(s)
  ChannelBlocks_3b2a84f1-0910-455c-8420-ec1d931a4331  // receive_pdo_parameter_RPDO2
  IO_1fe4c255-f970-4602-8183-e29f1a37e80e  // 1 Byte(s)
  IO_f76117aa-0616-4747-8f25-6d89972fd06d  // 1 Byte(s)
  IO_0ea4ff39-a97d-438f-bc89-279a651a34be  // 2 Byte(s)
  IO_46463791-502b-4132-94e5-2eb45fc9a8d2  // 4 Byte(s)
  ChannelBlocks_5d15d2f2-1d91-4b29-89c6-b4f2fd4c19d1  // transmit_pdo_parameter_TPDO1
  IO_11572021-aae5-43fa-8c81-8c65f5be2937  // 1 Byte(s)
  IO_11e39e64-b65e-428c-b496-34dc3f2bd81c  // 1 Byte(s)
  IO_66e25aa8-f219-450a-90ac-30608ca14490  // 1 Byte(s)
  IO_2e391c4d-0d29-4e3f-a3c2-c9202e5baf27  // 1 Byte(s)
  IO_d42ee03d-d42d-43fb-a7d7-544e10141c9a  // 4 Byte(s)
  ChannelBlocks_d8ea3532-8fe5-4ee2-8b30-17104c9e1a74  // transmit_pdo_parameter_TPDO2
  IO_c5531c87-81bc-40a7-b94b-1ab2f47d07bc  // 1 Byte(s)
  IO_3b70a104-6bda-4f1d-a8d3-184dd94ae2ef  // 1 Byte(s)
  IO_98bb85a8-f89b-4491-b75b-36770e484671  // 2 Byte(s)
  IO_18603d42-bde0-44ec-b6d7-79b9682289f6  // 4 Byte(s)
ServoUnit2 : FBD.Hilscher.COGenSlaveDTM.CMMS-ST (FHPP) (CMMS-ST_CAN_FHPP.eds) v0.0.0.0 (OrderNumber=CMMS_ST__FHPP___CMMS_ST_CAN_FHPP_eds_)  [CAN1 -> ServoUnit1.CAN2 (NodeNumber=13)]
  DtmId = 24ca3a76-7947-4b54-a270-430f39f0e1ad
  ChannelBlocks_f7b56e90-7f8b-4e90-815a-6c4dfc546ed7  // receive_pdo_parameter_RPDO1
  IO_9a79b520-762f-4938-959c-1673fd7573c4  // 1 Byte(s)
  IO_6f6dea46-2455-485a-94ad-83b3d498a592  // 1 Byte(s)
  IO_d006dc3e-8371-46dc-a683-50b710beabd8  // 1 Byte(s)
  IO_a5264c49-787e-4626-bff7-c2e1b2dd1289  // 1 Byte(s)
  IO_f44365d6-0f6b-46ff-a19d-db9847219f73  // 4 Byte(s)
  ChannelBlocks_ebb1fbf3-6661-4540-a5e3-a02181bc46a2  // receive_pdo_parameter_RPDO2
  IO_962121e9-a6d3-404e-abe5-8418554ba359  // 1 Byte(s)
  IO_f3f4d719-e6bc-434b-8025-6ba1cef229ee  // 1 Byte(s)
  IO_c1ece4da-ed7e-43ed-906d-7463e9429755  // 2 Byte(s)
  IO_cca085f9-9daf-4881-8b8f-ebd5b0e9fb28  // 4 Byte(s)
  ChannelBlocks_4914f731-ace5-4c21-b155-c44d73840a8b  // transmit_pdo_parameter_TPDO1
  IO_1f321ee5-e18e-49c4-b575-294241130312  // 1 Byte(s)
  IO_c8265208-a0c3-479d-8fa1-8b9fa156e66a  // 1 Byte(s)
  IO_dabdac96-5299-4b3b-accd-82906df4bf36  // 1 Byte(s)
  IO_883d6348-0267-4918-b7f4-9aca052a30fd  // 1 Byte(s)
  IO_79512acd-1801-4603-8a63-02ee5758af24  // 4 Byte(s)
  ChannelBlocks_b3aeed69-e232-4ad4-96ab-f421a44648fc  // transmit_pdo_parameter_TPDO2
  IO_28dfc721-11f9-4836-ae2e-81ac5ef2e3d2  // 1 Byte(s)
  IO_41e0f84a-fe01-4693-8d92-b2f94cad6525  // 1 Byte(s)
  IO_74d0d650-8c44-4949-92d7-296ea7dfe817  // 2 Byte(s)
  IO_6ebc7c61-af17-4b10-bee6-1b0b4320a898  // 4 Byte(s)
ServoUnit3 : FBD.Hilscher.COGenSlaveDTM.CMMS-ST (FHPP) (CMMS-ST_CAN_FHPP.eds) v0.0.0.0 (OrderNumber=CMMS_ST__FHPP___CMMS_ST_CAN_FHPP_eds_)  [CAN1 -> ServoUnit2.CAN2 (NodeNumber=15)]
  DtmId = 5020f104-a1e2-44d4-acb6-69c7e17304a7
  ChannelBlocks_d6aea6b7-799e-42d1-bb2c-abb3d7243e35  // receive_pdo_parameter_RPDO1
  IO_1edec1d8-fbb6-4ffc-8065-c09571833467  // 1 Byte(s)
  IO_e5602e7a-e0dc-4888-a40d-6a09cf17c6e9  // 1 Byte(s)
  IO_c34c2a29-a923-43e2-acfb-47e0a4efd83b  // 1 Byte(s)
  IO_8e27c422-e9dc-47bf-baf2-85f084dd8745  // 1 Byte(s)
  IO_f1eb85f8-4760-4688-933b-bf7fd4acfb4a  // 4 Byte(s)
  ChannelBlocks_9320c7e9-ebf6-45c0-b20f-8e1fd69b625e  // receive_pdo_parameter_RPDO2
  IO_20bbcb0d-084f-4822-8bde-928b78bc5ae1  // 1 Byte(s)
  IO_bf499093-88d7-4265-b01b-6f61ff49811d  // 1 Byte(s)
  IO_eb443335-35c4-401f-9a36-f292bfe6bbc6  // 2 Byte(s)
  IO_2b03c0a9-5f48-4dc4-a499-eefbdb215858  // 4 Byte(s)
  ChannelBlocks_9cb55215-4b1e-41d1-9087-a64961497188  // transmit_pdo_parameter_TPDO1
  IO_d2f6c6a5-7409-4d5f-8670-b92788f7687c  // 1 Byte(s)
  IO_d5532c33-4188-4f86-96bd-ae91e377d53b  // 1 Byte(s)
  IO_ef185e02-39e8-48ef-8fe3-fc49aa2e80d4  // 1 Byte(s)
  IO_10fc2cac-cd2e-4f93-886f-1acdfd1cf493  // 1 Byte(s)
  IO_35fcde1b-5957-49e4-a7c3-1ecdff961b11  // 4 Byte(s)
  ChannelBlocks_56541818-a82b-4211-915a-bba26b5d06a4  // transmit_pdo_parameter_TPDO2
  IO_e15f9eac-15fe-4db2-ac2b-eb41a4bc5c5b  // 1 Byte(s)
  IO_b64a1fd3-01ba-4664-a79a-20503f8bf38d  // 1 Byte(s)
  IO_4b91cf88-8a66-480e-b5b0-53a6a4a3d1e4  // 2 Byte(s)
  IO_7567258c-5454-45d0-a62f-76e1e24bd2cc  // 4 Byte(s)
ServoUnit4 : FBD.Hilscher.COGenSlaveDTM.CMMS-ST (FHPP) (CMMS-ST_CAN_FHPP.eds) v0.0.0.0 (OrderNumber=CMMS_ST__FHPP___CMMS_ST_CAN_FHPP_eds_)  [CAN1 -> ServoUnit3.CAN2 (NodeNumber=17)]
  DtmId = a34273b6-36be-4692-a4f2-d7fc8e714c63
  ChannelBlocks_9b6b0dcd-efb0-4e01-b60d-f1a2210800ab  // receive_pdo_parameter_RPDO1
  IO_72b4bdf3-ddcf-4d59-96f4-e77b92479034  // 1 Byte(s)
  IO_28d6c5ea-7894-4181-a2dd-c02c71614b69  // 1 Byte(s)
  IO_0a0a99bd-0a54-4de3-a355-4e34f248c40c  // 1 Byte(s)
  IO_0c63d19d-3bbb-4c5a-b3df-69e378063569  // 1 Byte(s)
  IO_d72d9506-6a6d-470a-95b9-72c2be7c6b4e  // 4 Byte(s)
  ChannelBlocks_8f802dff-d88f-4813-8999-1eadf24a71c8  // receive_pdo_parameter_RPDO2
  IO_04186658-edf4-456e-ae45-0e45d12bfb46  // 1 Byte(s)
  IO_51925c62-012b-4770-9bc1-e022595104c9  // 1 Byte(s)
  IO_394f25ff-c8b4-4b01-856b-71eccb60cd4a  // 2 Byte(s)
  IO_438dc71b-269e-4073-8cf1-927fb283052a  // 4 Byte(s)
  ChannelBlocks_32db9add-1d57-4f00-abc6-0aa464bc1857  // transmit_pdo_parameter_TPDO1
  IO_56facf51-be06-4162-8019-c9135e03ebd5  // 1 Byte(s)
  IO_c289eebf-ff75-4115-ae67-bb220dd48802  // 1 Byte(s)
  IO_d8c5064e-3c4b-4b83-a08c-9356c72a7307  // 1 Byte(s)
  IO_3c253702-47c6-475a-b5a9-f2037096e21d  // 1 Byte(s)
  IO_20db09f5-c500-42c7-9670-06e013c1e1a7  // 4 Byte(s)
  ChannelBlocks_d3f68f18-3b23-4a83-8432-9608af0a8a6d  // transmit_pdo_parameter_TPDO2
  IO_6d3eccf2-412e-4869-bbf7-3d5ee19acd1b  // 1 Byte(s)
  IO_790cfb60-51d9-4129-97dc-1306fc7ae3f2  // 1 Byte(s)
  IO_b3acf3a2-48d5-43e6-9414-918042759147  // 2 Byte(s)
  IO_3bd5798b-ff23-498c-b349-786a6d395acf  // 4 Byte(s)
ServoUnit5 : FBD.Hilscher.COGenSlaveDTM.CMMS-ST (FHPP) (CMMS-ST_CAN_FHPP.eds) v0.0.0.0 (OrderNumber=CMMS_ST__FHPP___CMMS_ST_CAN_FHPP_eds_)  [CAN1 -> ServoUnit4.CAN2 (NodeNumber=19)]
  DtmId = dddd2ea4-72f4-41ff-b4f0-61cd90decc37
  ChannelBlocks_b2a47bf8-6451-4bcc-8048-7b48c7bb103f  // receive_pdo_parameter_RPDO1
  IO_042c1306-50b9-4a2e-af5d-07a155835bcd  // 1 Byte(s)
  IO_f95a7d75-ca02-4e9e-816a-ea6511c469e3  // 1 Byte(s)
  IO_1e96aa95-6ac6-466c-8375-caaf705f7563  // 1 Byte(s)
  IO_aec588cb-3200-4f30-8b62-ac89dcc3257c  // 1 Byte(s)
  IO_58883095-a84a-422e-9e67-136805d76ca8  // 4 Byte(s)
  ChannelBlocks_a1a16dd9-e4cc-4529-a01a-5b4485273169  // receive_pdo_parameter_RPDO2
  IO_201606b6-99f1-4817-9c48-41f53bc3413e  // 1 Byte(s)
  IO_2354511c-5730-4c6f-b022-568f79be2817  // 1 Byte(s)
  IO_c8bb1aac-b248-4641-bbd6-8c43b71ac324  // 2 Byte(s)
  IO_d370564a-a8fc-4719-b186-8a9189a9ffea  // 4 Byte(s)
  ChannelBlocks_e43a4828-9791-4349-8756-650c10531e77  // transmit_pdo_parameter_TPDO1
  IO_36510441-71fd-4c1f-b6c2-76242bff5ce4  // 1 Byte(s)
  IO_79cbc5fc-c8bb-4913-a882-52f30785010e  // 1 Byte(s)
  IO_b825f711-752e-49af-8167-44fb10692939  // 1 Byte(s)
  IO_1b5ef188-911d-4237-8649-bcb55827c28f  // 1 Byte(s)
  IO_271c16a8-7d34-4570-b9da-a54ad545dc98  // 4 Byte(s)
  ChannelBlocks_4bc3a0fa-b3a3-4bfd-a8a2-920f368d3016  // transmit_pdo_parameter_TPDO2
  IO_86bcbf9c-29d2-4335-9fed-c91db8038985  // 1 Byte(s)
  IO_57d457d1-12c3-49a6-a86f-0825d01c51a9  // 1 Byte(s)
  IO_20155857-eeeb-462d-bfc0-4988759b86e8  // 2 Byte(s)
  IO_2c2b4482-8124-4308-9cc1-4542e1d09207  // 4 Byte(s)
ServoUnit6 : FBD.Hilscher.COGenSlaveDTM.CMMS-ST (FHPP) (CMMS-ST_CAN_FHPP.eds) v0.0.0.0 (OrderNumber=CMMS_ST__FHPP___CMMS_ST_CAN_FHPP_eds_)  [CAN1 -> ServoUnit5.CAN2 (NodeNumber=21)]
  DtmId = 34532c5a-2d2e-4b03-9bc7-8850a67d2130
  ChannelBlocks_014097cd-8ac2-4333-968e-92bf850f96c7  // receive_pdo_parameter_RPDO1
  IO_c267876c-3ee7-44dc-8baa-c6297e9e396c  // 1 Byte(s)
  IO_36021023-e771-4991-883d-6380b1a1f41a  // 1 Byte(s)
  IO_688c0272-c617-43a2-a663-be775dbde0f8  // 1 Byte(s)
  IO_226f68f9-27e0-4731-8149-1088403f2aa7  // 1 Byte(s)
  IO_475b073e-e09b-44ab-98ad-44bf06c853b7  // 4 Byte(s)
  ChannelBlocks_3bdc7835-cce4-4e3c-80e4-686c9cceda84  // receive_pdo_parameter_RPDO2
  IO_f518c910-137c-4fa1-9bbd-8b61a6f4dc37  // 1 Byte(s)
  IO_83fec91e-204c-46c4-8cbb-fc5a6f6a1236  // 1 Byte(s)
  IO_3dba2bb8-d2c7-4cc6-b000-f3edc82f1d62  // 2 Byte(s)
  IO_abd3ffe8-6828-47eb-9432-002f410b4f4c  // 4 Byte(s)
  ChannelBlocks_fac5cb02-686b-4465-b0f6-ed87e816fcc1  // transmit_pdo_parameter_TPDO1
  IO_b8addc99-4bdf-4daf-9b2c-58a510851fe2  // 1 Byte(s)
  IO_983db230-7526-481f-986f-203a5a9ca751  // 1 Byte(s)
  IO_98bb3a7b-510b-4093-ba63-1e745c7b40f2  // 1 Byte(s)
  IO_e9279d78-9754-4347-8dc9-ef642c374f5c  // 1 Byte(s)
  IO_b0cd985d-e990-4e0b-aba7-7a18131281a8  // 4 Byte(s)
  ChannelBlocks_df8160ba-0a2a-48d2-9cb1-1acc8398b25d  // transmit_pdo_parameter_TPDO2
  IO_a8478a33-7798-4d6d-aa16-4210a747f91f  // 1 Byte(s)
  IO_b2251cb0-e264-414f-b404-bba09d574283  // 1 Byte(s)
  IO_e3a1305f-f38b-429b-af16-593b6c6e717a  // 2 Byte(s)
  IO_f7517dfb-5583-4d37-b2a5-136d0ab4f222  // 4 Byte(s)
ServoUnit7 : FBD.Hilscher.COGenSlaveDTM.CMMS-ST (FHPP) (CMMS-ST_CAN_FHPP.eds) v0.0.0.0 (OrderNumber=CMMS_ST__FHPP___CMMS_ST_CAN_FHPP_eds_)  [CAN1 -> ServoUnit6.CAN2 (NodeNumber=23)]
  DtmId = 5fc7343d-0ed6-405b-8d95-2105416229d2
  ChannelBlocks_5eb8554f-0563-4c22-9e94-801e002a6495  // receive_pdo_parameter_RPDO1
  IO_d9adffc7-890e-4265-9bdb-82d5b69f6456  // 1 Byte(s)
  IO_2e912434-e4e4-4d4a-b4fa-36df2f75fcf2  // 1 Byte(s)
  IO_9388c441-335f-4d87-b598-0a50b2084254  // 1 Byte(s)
  IO_164f78f4-70d7-4b4b-bc6f-9586e17082c1  // 1 Byte(s)
  IO_e78b788c-81d5-4b1d-98e5-c6d7e026460a  // 4 Byte(s)
  ChannelBlocks_3e361ac6-f3cb-4ba3-b415-3a103ca45a69  // receive_pdo_parameter_RPDO2
  IO_9cb82a6f-f4cc-462d-887a-0b28df0f1edf  // 1 Byte(s)
  IO_34740f43-5725-44c3-a83e-7975d3695ec9  // 1 Byte(s)
  IO_0528aa5b-7607-4c2d-b848-d1a5daa0e49e  // 2 Byte(s)
  IO_8231ce7c-6fd5-4cbb-a00a-fee86b9cdc1d  // 4 Byte(s)
  ChannelBlocks_d60dd0ff-9d93-4d0f-bb52-2b4e21ac8004  // transmit_pdo_parameter_TPDO1
  IO_7fb01a7b-c935-4f43-83d9-e868a22cc3e6  // 1 Byte(s)
  IO_968dbf1f-6d23-4d5d-8859-f1edde25f2cd  // 1 Byte(s)
  IO_a53445b8-d39c-4e80-a914-5ed1505b6e51  // 1 Byte(s)
  IO_3387e47b-ce9f-48f4-b2a7-57df4d28f3b6  // 1 Byte(s)
  IO_f90b1322-f687-48e9-96dd-69ca3767db28  // 4 Byte(s)
  ChannelBlocks_3b12632d-dcd6-43d4-b35c-fa14bea89791  // transmit_pdo_parameter_TPDO2
  IO_0b26b99f-e93e-4bcb-b486-e64ae01993d4  // 1 Byte(s)
  IO_3e79ad31-592d-4325-81b2-a2d015b077a7  // 1 Byte(s)
  IO_c8079b08-2069-4517-97c1-607e64962062  // 2 Byte(s)
  IO_561002b7-5777-4273-b568-5d73c2089a36  // 4 Byte(s)
ServoUnit8 : FBD.Hilscher.COGenSlaveDTM.CMMS-ST (FHPP) (CMMS-ST_CAN_FHPP.eds) v0.0.0.0 (OrderNumber=CMMS_ST__FHPP___CMMS_ST_CAN_FHPP_eds_)  [CAN1 -> ServoUnit7.CAN2 (NodeNumber=25)]
  DtmId = 4ec47f7c-6edc-42d7-a472-79fd813b55ba
  ChannelBlocks_fe87a98e-0f02-4bb8-8635-11464382610f  // receive_pdo_parameter_RPDO1
  IO_fbb65677-c766-47a3-8ac3-1a8fa791d6b4  // 1 Byte(s)
  IO_e4962899-6911-4df9-b9a1-55919f7208f7  // 1 Byte(s)
  IO_2c3a640c-870f-4d1e-8044-cc15a12cc6ca  // 1 Byte(s)
  IO_d13546d0-3934-4e2d-879b-8538331d70bb  // 1 Byte(s)
  IO_c6bf2520-d47f-437d-ab21-7c0fd25d66ca  // 4 Byte(s)
  ChannelBlocks_d67310ef-a431-4a4f-bcab-ccee4ed7fe25  // receive_pdo_parameter_RPDO2
  IO_1011048c-ae09-4a9e-9577-ef76f6e644eb  // 1 Byte(s)
  IO_b57aba91-06bf-44d7-8d0e-3bb4fc99e55d  // 1 Byte(s)
  IO_a1c9e2d8-dd8a-48e5-86e3-cae28a455347  // 2 Byte(s)
  IO_f6bd3884-971a-46b4-9642-246530a3e1b5  // 4 Byte(s)
  ChannelBlocks_d7a9a873-866e-4503-8882-9bef2a1b5558  // transmit_pdo_parameter_TPDO1
  IO_741aed39-42ce-401e-bec2-763fb2a9c994  // 1 Byte(s)
  IO_e87c71ab-78f0-45a2-a3f3-b6a76e617efc  // 1 Byte(s)
  IO_800b70cc-9aea-40d1-bc25-84b4df11980d  // 1 Byte(s)
  IO_895030f8-d70f-46ed-96b2-1facfe63d131  // 1 Byte(s)
  IO_e1d0605e-273c-497d-81da-54f8edf83c62  // 4 Byte(s)
  ChannelBlocks_916496bc-f4e5-4235-8735-bf956dd8cf6a  // transmit_pdo_parameter_TPDO2
  IO_ff84d874-16ff-4916-826a-b20360c3d884  // 1 Byte(s)
  IO_6aaf0cc2-08a4-4618-a070-07df5d000b7c  // 1 Byte(s)
  IO_1a7e0e65-21fc-47d8-ac29-fe06e8a3c122  // 2 Byte(s)
  IO_42eb6130-3075-4df7-a7f4-ff76522d1257  // 4 Byte(s)
ServoUnit9 : FBD.Hilscher.COGenSlaveDTM.CMMS-ST (FHPP) (CMMS-ST_CAN_FHPP.eds) v0.0.0.0 (OrderNumber=CMMS_ST__FHPP___CMMS_ST_CAN_FHPP_eds_)  [CAN1 -> ServoUnit8.CAN2 (NodeNumber=27)]
  DtmId = 671d1f85-f1e9-4568-b545-12b1f0c7e482
  ChannelBlocks_dd0a8c76-d38b-4773-995a-5e9fb78888d0  // receive_pdo_parameter_RPDO1
  IO_aa9e0205-39f5-406a-a6b0-77c12f17dcb4  // 1 Byte(s)
  IO_ee854bcf-83f6-4455-afcc-d544571dd1de  // 1 Byte(s)
  IO_4d133417-e236-4804-8198-80d1e1dd82d7  // 1 Byte(s)
  IO_e1b26244-7bea-4eed-ae3b-03f85235d93d  // 1 Byte(s)
  IO_aac6794d-a446-4c43-8f5b-09daea610a2e  // 4 Byte(s)
  ChannelBlocks_9728e1b6-f62c-4575-967e-0388b8133728  // receive_pdo_parameter_RPDO2
  IO_93cf6017-a56e-4696-bf1c-3441967dc200  // 1 Byte(s)
  IO_e6ed09c3-5c56-4f3b-b18f-de59b491be24  // 1 Byte(s)
  IO_436a10a5-4a5f-4913-a60b-a38dd568ab0b  // 2 Byte(s)
  IO_2c1050d5-aab6-491d-92b4-a032e5286b99  // 4 Byte(s)
  ChannelBlocks_5a5b70af-9560-4f35-be0c-1f7e75638ebb  // transmit_pdo_parameter_TPDO1
  IO_c2889cc6-41fd-42a5-8e16-53288c27a8a8  // 1 Byte(s)
  IO_dc6f2658-764b-4710-a3b8-111945dc1cee  // 1 Byte(s)
  IO_d7331c01-ffe8-4a85-b933-3f75d1175aa3  // 1 Byte(s)
  IO_f5380f58-a010-42a6-ac55-831522e03977  // 1 Byte(s)
  IO_e9dff24f-4577-467f-9178-0208c2a626d8  // 4 Byte(s)
  ChannelBlocks_88f7015e-866a-4655-b200-07d27eb34ebc  // transmit_pdo_parameter_TPDO2
  IO_2081798b-f002-47cb-94a9-62caf60cee85  // 1 Byte(s)
  IO_38dcf81d-0990-463e-9b03-7b23085dfe67  // 1 Byte(s)
  IO_23f2c857-c315-4d74-b26a-a1c481f7a1c7  // 2 Byte(s)
  IO_4be5187b-eac9-42d4-82d3-71e8956ff4e4  // 4 Byte(s)
X20BC0083 : X20BC0083 v2.1.0.0  [PLK1 -> X20CP1585.IF3 (NodeNumber=1); PLK2 -> X20BC0083b.PLK1 (NodeNumber=1); SL -> BU_0-1.SL1]
  Supervision = off
X20BC0083a : X20BC0083 v2.1.0.0  [PLK1 -> X20BC0083e.PLK2 (NodeNumber=6); SL -> MBU.SL1]
  Supervision = off
X20BC0083b : X20BC0083 v2.1.0.0  [PLK1 -> X20BC0083.PLK2 (NodeNumber=2); PLK2 -> X20BC0083c.PLK1 (NodeNumber=2); SL -> BU_2-3.SL1]
  Supervision = off
X20BC0083c : X20BC0083 v2.1.0.0  [PLK1 -> X20BC0083b.PLK2 (NodeNumber=3); PLK2 -> X20BC0083d.PLK1 (NodeNumber=3); SL -> BU_4-5.SL1]
  Supervision = off
X20BC0083d : X20BC0083 v2.1.0.0  [PLK1 -> X20BC0083c.PLK2 (NodeNumber=4); PLK2 -> X20BC0083e.PLK1 (NodeNumber=4); SL -> BU_6-7.SL1]
  Supervision = off
X20BC0083e : X20BC0083 v2.1.0.0  [PLK1 -> X20BC0083d.PLK2 (NodeNumber=5); PLK2 -> X20BC0083a.PLK1 (NodeNumber=5); SL -> BU_8-9.SL1]
  Supervision = off
X20BM11 : X20BM11 v1.0.0.0  [X2X1 -> BU_0-1.IF1]
X20BM11a : X20BM11 v1.0.0.0  [X2X1 -> X20BM11f.X2X2]
X20BM11b : X20BM11 v1.0.0.0  [X2X1 -> X20BM11.X2X2]
X20BM11c : X20BM11 v1.0.0.0  [X2X1 -> X20BM11a.X2X2]
X20BM11d : X20BM11 v1.0.0.0  [X2X1 -> X20BM11e.X2X2]
X20BM11e : X20BM11 v1.0.0.0  [X2X1 -> X20BM11c.X2X2]
X20BM11f : X20BM11 v1.0.0.0  [X2X1 -> X20CP1585.IF6]
X20BM11g : X20BM11 v1.0.0.0  [X2X1 -> MBU.IF1]
X20BM11h : X20BM11 v1.0.0.0  [X2X1 -> X20BM11g.X2X2]
X20BM11i : X20BM11 v1.0.0.0  [X2X1 -> BU_2-3.IF1]
X20BM11j : X20BM11 v1.0.0.0  [X2X1 -> BU_4-5.IF1]
X20BM11k : X20BM11 v1.0.0.0  [X2X1 -> BU_6-7.IF1]
X20BM11l : X20BM11 v1.0.0.0  [X2X1 -> BU_8-9.IF1]
X20BM11m : X20BM11 v1.0.0.0  [X2X1 -> X20BM11i.X2X2]
X20BM11n : X20BM11 v1.0.0.0  [X2X1 -> X20BM11j.X2X2]
X20BM11o : X20BM11 v1.0.0.0  [X2X1 -> X20BM11k.X2X2]
X20BM11p : X20BM11 v1.0.0.0  [X2X1 -> X20BM11l.X2X2]
X20CP1585 : X20CP1585 v1.0.4.0
  Connector IF2:
    ActivateDevice = 1
    EthInterfaceRedundant = 0
    HostName = if2-themagnifica_semp
    Mode = Manual
    InternetAddress = 192.168.40.155
    SubnetMask = 255.255.255.0
    Vnc1
    VncVcObjectName1 = BU_Gui
    VncKeyMappingFile1 = VC\PS2-Keyboard.dis
    Vnc2
    VncVcObjectName2 = Mobile
    VncKeyMappingFile2 = VC\PS2-Keyboard1.dis
    VncPortNumber2 = 5901
  Connector IF3:
    EplInterfaceRedundant = 0
    EplHostName = if3-themagnifica_semp
    EplEthInterfaceRedundant = 0
    HostName = if3-eth-themagnifica_semp
  Connector IF6:
    CycleTime = 1000
    BusLength = 100
    Stations = 8
  ConfigurationID = The_Magnifica_v0157_X20
  RebootReset = 1
  TimerDeviceType = SWIOTIMER
  CyclicTaskClassCount = 5
  Cyclic1Duration = 1000
  Cyclic1Tolerance = 0
  Cyclic1Output = 1
  Cyclic2Duration = 5000
  Cyclic2Tolerance = 0
  Cyclic3Duration = 50000
  Cyclic3Tolerance = 0
  Cyclic4Duration = 100000
  Cyclic4Tolerance = 0
  Cyclic5Duration = 10000
  Cyclic5Tolerance = 30000000
  Cyclic6Duration = 500000
  Cyclic6Tolerance = 500000
  Cyclic7Duration = 1000000
  Cyclic7Tolerance = 1000000
  Cyclic8Duration = 10000
  Cyclic8Tolerance = 30000000
  TimeZone = 140
  ActivateDaylightSavingTime = 1
  ActivateSntp = 1
  SntpcServAddr1 = time.windows.com
  SntpcServAddr2 = time.windows.com
  EthernetHostName = themagnifica_semp
  EthernetDefaultGateway = 192.168.40.1
  ActivateDns = 1
  GetDnsFromDhcp = 2
  FtpUser1
  FtpUsername1 = plc
  FtpUserPassword1 = WAJG592WMMVamzkpViOP3PaAh6yYa8m5godAftJLDBo=
  FtpUserSalt1 = mpJEyBZ7
  FTPAccessRight1 = 0
  ActivateOpcUa = 1
  OpcUaAnonymous = 1
  OpcUaMaxSubsItemQueueSize = 10000
X20IF1041_1 : X20IF1041-1 v1.1.1.1  [SS -> X20CP1585.SS1]
  Connector IF1:
    DtmRef = FBDIF.Hilscher.COMDtmNX.NETX 100 CO/COM
    DtmId = 71bebc67-7576-41f1-883e-778b88cef510
  ConfigFile = X20IF1041_1.dtm
  ConfigModule = asnxdb2
  ConfigUID = 1009496404
X20PS9400 : X20PS9400 v1.0.2.1  [SS1 -> X20TB12a.SS; PS -> BU_0-1.PS1]
  Supervision = off
X20PS9400a : X20PS9400 v1.0.2.1  [SS1 -> X20TB12h.SS; PS -> MBU.PS1]
  Supervision = off
X20PS9400b : X20PS9400 v1.0.2.1  [SS1 -> X20TB12k.SS; PS -> BU_2-3.PS1]
  Supervision = off
X20PS9400c : X20PS9400 v1.0.2.1  [SS1 -> X20TB12l.SS; PS -> BU_4-5.PS1]
  Supervision = off
X20PS9400d : X20PS9400 v1.0.2.1  [SS1 -> X20TB12m.SS; PS -> BU_6-7.PS1]
  Supervision = off
X20PS9400e : X20PS9400 v1.0.2.1  [SS1 -> X20TB12n.SS; PS -> BU_8-9.PS1]
  Supervision = off
X20TB12 : X20TB12 v1.0.0.0
X20TB12a : X20TB12 v1.0.0.0
X20TB12b : X20TB12 v1.0.0.0
X20TB12c : X20TB12 v1.0.0.0
X20TB12d : X20TB12 v1.0.0.0
X20TB12e : X20TB12 v1.0.0.0
X20TB12f : X20TB12 v1.0.0.0
X20TB12g : X20TB12 v1.0.0.0
X20TB12h : X20TB12 v1.0.0.0
X20TB12i : X20TB12 v1.0.0.0
X20TB12j : X20TB12 v1.0.0.0
X20TB12k : X20TB12 v1.0.0.0
X20TB12l : X20TB12 v1.0.0.0
X20TB12m : X20TB12 v1.0.0.0
X20TB12n : X20TB12 v1.0.0.0
X20TB12o : X20TB12 v1.0.0.0
X20TB12p : X20TB12 v1.0.0.0
X20TB12q : X20TB12 v1.0.0.0
X20TB12r : X20TB12 v1.0.0.0
X20TB12s : X20TB12 v1.0.0.0
X20TB12t : X20TB12 v1.0.0.0
X20TB12u : X20TB12 v1.0.0.0
X20TB12v : X20TB12 v1.0.0.0
```

### IoMap.iom - X20CP1585/IoMap.iom
```iecst
(********************************************************************
 * COPYRIGHT --
 ********************************************************************
 * File: IoMap.iom
 * Author: jorkes
 * Created: July 07, 2014
 ********************************************************************
 * IO mapping file
 ********************************************************************)
VAR_CONFIG
	Cyclic#1.MBU.in_bMainBeltSensor1 AT %IX."in_MCU".DigitalInput01;
	Cyclic#1.MBU.in_bMainBeltSensor2 AT %IX."in_MCU".DigitalInput02;
	Cyclic#1.MCU.typIN.bEncPuls1 AT %IX."in_MCU".DigitalInput03;
	Cyclic#3.MCU.typIN.bJog AT %IX."in_MCU".DigitalInput07;
	Cyclic#3.MCU.typIN.bDoorOpen AT %IX."in_MCU".DigitalInput08;
	Cyclic#3.MCU.typIN.bEmergencyStop AT %IX."in_MCU".DigitalInput09;
	Cyclic#3.MCU.typIN.bServiceMode AT %IX."in_MCU".DigitalInput10;
	Cyclic#3.MCU.typIN.bAirpressure AT %IX."in_MCU".DigitalInput11;
	Cyclic#1.MCU.typOUT.bCamTrigger1 AT %QX."out_MCU_0".DigitalOutput01;
	Cyclic#1.MCU.typOUT.bCamTrigger2 AT %QX."out_MCU_0".DigitalOutput03;
	Cyclic#1.MCU.typOUT.bLightTrigger2 AT %QX."out_MCU_0".DigitalOutput04;
	Cyclic#1.MCU.typOUT.bCamTrigger3 AT %QX."out_MCU_0".DigitalOutput05;
	Cyclic#1.MCU.typOUT.bLightTrigger3 AT %QX."out_MCU_0".DigitalOutput06;
	Cyclic#1.MCU.typOUT.bCamTrigger4 AT %QX."out_MCU_0".DigitalOutput07;
	Cyclic#1.MCU.typOUT.bLightTrigger4 AT %QX."out_MCU_0".DigitalOutput08;
	Cyclic#1.RU.typOUT.bActivateGripper AT %QX."out_MCU_0".DigitalOutput12;
	Cyclic#1.BU[0].typOUT.bActivateGripper AT %QX."out_MCU_1".DigitalOutput01;
	Cyclic#1.BU[1].typOUT.bActivateGripper AT %QX."out_MCU_1".DigitalOutput02;
	Cyclic#1.BU[2].typOUT.bActivateGripper AT %QX."out_MCU_1".DigitalOutput03;
	Cyclic#1.BU[3].typOUT.bActivateGripper AT %QX."out_MCU_1".DigitalOutput04;
	Cyclic#1.BU[4].typOUT.bActivateGripper AT %QX."out_MCU_1".DigitalOutput05;
	Cyclic#1.BU[5].typOUT.bActivateGripper AT %QX."out_MCU_1".DigitalOutput06;
	Cyclic#1.BU[6].typOUT.bActivateGripper AT %QX."out_MCU_1".DigitalOutput07;
	Cyclic#1.BU[7].typOUT.bActivateGripper AT %QX."out_MCU_1".DigitalOutput08;
	Cyclic#1.BU[8].typOUT.bActivateGripper AT %QX."out_MCU_1".DigitalOutput09;
	Cyclic#1.BU[9].typOUT.bActivateGripper AT %QX."out_MCU_1".DigitalOutput10;
	Cyclic#3.MCU.typOUT.bGreenLight AT %QX."out_MCU_1".DigitalOutput11;
	Cyclic#3.MCU.typOUT.bRedLight AT %QX."out_MCU_1".DigitalOutput12;
	Cyclic#1.BU[0].typOUT.bBunchGripper AT %QX."out_MCU_2".DigitalOutput01;
	Cyclic#1.BU[1].typOUT.bBunchGripper AT %QX."out_MCU_2".DigitalOutput02;
	Cyclic#1.BU[2].typOUT.bBunchGripper AT %QX."out_MCU_2".DigitalOutput03;
	Cyclic#1.BU[3].typOUT.bBunchGripper AT %QX."out_MCU_2".DigitalOutput04;
	Cyclic#1.BU[4].typOUT.bBunchGripper AT %QX."out_MCU_2".DigitalOutput05;
	Cyclic#1.BU[5].typOUT.bBunchGripper AT %QX."out_MCU_2".DigitalOutput06;
	Cyclic#1.BU[6].typOUT.bBunchGripper AT %QX."out_MCU_2".DigitalOutput07;
	Cyclic#1.BU[7].typOUT.bBunchGripper AT %QX."out_MCU_2".DigitalOutput08;
	Cyclic#1.BU[8].typOUT.bBunchGripper AT %QX."out_MCU_2".DigitalOutput09;
	Cyclic#1.BU[9].typOUT.bBunchGripper AT %QX."out_MCU_2".DigitalOutput10;
	Cyclic#1.MCU.typOUT.bBuzzer AT %QX."out_MCU_3".DigitalOutput09;
	Cyclic#3.MCU.typOUT.bGreenLight AT %QX."out_MCU_3".DigitalOutput07;
	Cyclic#3.MCU.typOUT.bRedLight AT %QX."out_MCU_3".DigitalOutput08;
	Cyclic#3.MCU.typOUT.bMachineShutDown AT %QX."out_MCU_3".DigitalOutput10;
	Cyclic#3.MCU.typOUT.bResetDoorOpen AT %QX."out_MCU_3".DigitalOutput11;
	Cyclic#3.MCU.typOUT.bResetEmergencyStop AT %QX."out_MCU_3".DigitalOutput12;
	Cyclic#3.BU[0].typIN.bElevatorUp AT %IX."in_BU_0-1".DigitalInput01;
	Cyclic#3.BU[1].typIN.bElevatorUp AT %IX."in_BU_0-1".DigitalInput02;
	Cyclic#2.BU[0].typIN.bElevatorMid AT %IX."in_BU_0-1".DigitalInput03;
	Cyclic#2.BU[1].typIN.bElevatorMid AT %IX."in_BU_0-1".DigitalInput04;
	Cyclic#2.BU[0].typIN.bElevatorDown AT %IX."in_BU_0-1".DigitalInput05;
	Cyclic#2.BU[1].typIN.bElevatorDown AT %IX."in_BU_0-1".DigitalInput06;
	Cyclic#3.BU[1].typIN.bTestUnit AT %IX."in_BU_0-1".DigitalInput08;
	Cyclic#3.BU[0].typIN.bTestUnit AT %IX."in_BU_0-1".DigitalInput07;
	Cyclic#3.BU[0].typIN.bOnline AT %IX."in_BU_0-1".ModuleOk;
	Cyclic#3.BU[0].typOUT.bOnline AT %IX."out_BU_0-1".ModuleOk;
	Cyclic#1.BU[0].typOUT.bElevator AT %QX."out_BU_0-1".DigitalOutput01;
	Cyclic#1.BU[1].typOUT.bElevator AT %QX."out_BU_0-1".DigitalOutput02;
	Cyclic#1.BU[0].typOUT.bReleaseGripper AT %QX."out_BU_0-1".DigitalOutput03;
	Cyclic#1.BU[1].typOUT.bReleaseGripper AT %QX."out_BU_0-1".DigitalOutput04;
	Cyclic#3.BU[0].typOUT.bStopServo AT %QX."out_BU_0-1".DigitalOutput05;
	Cyclic#3.BU[1].typOUT.bStopServo AT %QX."out_BU_0-1".DigitalOutput06;
	Cyclic#3.BU[0].typOUT.bEndStageServo AT %QX."out_BU_0-1".DigitalOutput07;
	Cyclic#3.BU[1].typOUT.bEndStageServo AT %QX."out_BU_0-1".DigitalOutput08;
	Cyclic#3.BU[0].typOUT.bEnableServo AT %QX."out_BU_0-1".DigitalOutput09;
	Cyclic#3.BU[1].typOUT.bEnableServo AT %QX."out_BU_0-1".DigitalOutput10;
	Cyclic#1.BU[0].bAddFlower AT %QX."out_BU_0-1".DigitalOutput11; (*24 VDC / 0.5 A, source (test add active)*)
	Cyclic#1.BU[1].bAddFlower AT %QX."out_BU_0-1".DigitalOutput12; (*24 VDC / 0.5 A, source (Test add active)*)
	Cyclic#1.BU[2].typIN.bElevatorUp AT %IX."in_BU_2-3".DigitalInput01;
	Cyclic#1.BU[3].typIN.bElevatorUp AT %IX."in_BU_2-3".DigitalInput02;
	Cyclic#1.BU[2].typIN.bElevatorMid AT %IX."in_BU_2-3".DigitalInput03;
	Cyclic#1.BU[3].typIN.bElevatorMid AT %IX."in_BU_2-3".DigitalInput04;
	Cyclic#1.BU[2].typIN.bElevatorDown AT %IX."in_BU_2-3".DigitalInput05;
	Cyclic#1.BU[3].typIN.bElevatorDown AT %IX."in_BU_2-3".DigitalInput06;
	Cyclic#1.BU[2].typIN.bTestUnit AT %IX."in_BU_2-3".DigitalInput07;
	Cyclic#1.BU[3].typIN.bTestUnit AT %IX."in_BU_2-3".DigitalInput08;
	Cyclic#3.BU[2].typIN.bOnline AT %IX."in_BU_0-1".ModuleOk;
	Cyclic#3.BU[2].typOUT.bOnline AT %IX."out_BU_0-1".ModuleOk;
	Cyclic#1.BU[2].typOUT.bElevator AT %QX."out_BU_2-3".DigitalOutput01;
	Cyclic#1.BU[3].typOUT.bElevator AT %QX."out_BU_2-3".DigitalOutput02;
	Cyclic#1.BU[2].typOUT.bReleaseGripper AT %QX."out_BU_2-3".DigitalOutput03;
	Cyclic#1.BU[3].typOUT.bReleaseGripper AT %QX."out_BU_2-3".DigitalOutput04;
	Cyclic#3.BU[2].typOUT.bStopServo AT %QX."out_BU_2-3".DigitalOutput05;
	Cyclic#3.BU[3].typOUT.bStopServo AT %QX."out_BU_2-3".DigitalOutput06;
	Cyclic#3.BU[2].typOUT.bEndStageServo AT %QX."out_BU_2-3".DigitalOutput07;
	Cyclic#3.BU[3].typOUT.bEndStageServo AT %QX."out_BU_2-3".DigitalOutput08;
	Cyclic#3.BU[2].typOUT.bEnableServo AT %QX."out_BU_2-3".DigitalOutput09;
	Cyclic#3.BU[3].typOUT.bEnableServo AT %QX."out_BU_2-3".DigitalOutput10;
	Cyclic#1.BU[2].bAddFlower AT %QX."out_BU_2-3".DigitalOutput11; (*24 VDC / 0.5 A, source (test add active)*)
	Cyclic#1.BU[3].bAddFlower AT %QX."out_BU_2-3".DigitalOutput12; (*24 VDC / 0.5 A, source (Test add active)*)
	Cyclic#1.BU[4].typIN.bElevatorUp AT %IX."in_BU_4-5".DigitalInput01;
	Cyclic#1.BU[5].typIN.bElevatorUp AT %IX."in_BU_4-5".DigitalInput02;
	Cyclic#1.BU[4].typIN.bElevatorMid AT %IX."in_BU_4-5".DigitalInput03;
	Cyclic#1.BU[5].typIN.bElevatorMid AT %IX."in_BU_4-5".DigitalInput04;
	Cyclic#1.BU[4].typIN.bElevatorDown AT %IX."in_BU_4-5".DigitalInput05;
	Cyclic#1.BU[5].typIN.bElevatorDown AT %IX."in_BU_4-5".DigitalInput06;
	Cyclic#1.BU[4].typIN.bTestUnit AT %IX."in_BU_4-5".DigitalInput07;
	Cyclic#1.BU[5].typIN.bTestUnit AT %IX."in_BU_4-5".DigitalInput08;
	Cyclic#3.BU[4].typIN.bOnline AT %IX."in_BU_0-1".ModuleOk;
	Cyclic#3.BU[4].typOUT.bOnline AT %IX."out_BU_0-1".ModuleOk;
	Cyclic#1.BU[4].typOUT.bElevator AT %QX."out_BU_4-5".DigitalOutput01;
	Cyclic#1.BU[5].typOUT.bElevator AT %QX."out_BU_4-5".DigitalOutput02;
	Cyclic#1.BU[4].typOUT.bReleaseGripper AT %QX."out_BU_4-5".DigitalOutput03;
	Cyclic#1.BU[5].typOUT.bReleaseGripper AT %QX."out_BU_4-5".DigitalOutput04;
	Cyclic#3.BU[4].typOUT.bStopServo AT %QX."out_BU_4-5".DigitalOutput05;
	Cyclic#3.BU[5].typOUT.bStopServo AT %QX."out_BU_4-5".DigitalOutput06;
	Cyclic#3.BU[4].typOUT.bEndStageServo AT %QX."out_BU_4-5".DigitalOutput07;
	Cyclic#3.BU[5].typOUT.bEndStageServo AT %QX."out_BU_4-5".DigitalOutput08;
	Cyclic#3.BU[4].typOUT.bEnableServo AT %QX."out_BU_4-5".DigitalOutput09;
	Cyclic#3.BU[5].typOUT.bEnableServo AT %QX."out_BU_4-5".DigitalOutput10;
	Cyclic#1.BU[4].bAddFlower AT %QX."out_BU_4-5".DigitalOutput11; (*24 VDC / 0.5 A, source (test add active)*)
	Cyclic#1.BU[5].bAddFlower AT %QX."out_BU_4-5".DigitalOutput12; (*24 VDC / 0.5 A, source (Test add active)*)
	Cyclic#1.BU[6].typIN.bElevatorUp AT %IX."in_BU_6-7".DigitalInput01;
	Cyclic#1.BU[7].typIN.bElevatorUp AT %IX."in_BU_6-7".DigitalInput02;
	Cyclic#1.BU[6].typIN.bElevatorMid AT %IX."in_BU_6-7".DigitalInput03;
	Cyclic#1.BU[7].typIN.bElevatorMid AT %IX."in_BU_6-7".DigitalInput04;
	Cyclic#1.BU[6].typIN.bElevatorDown AT %IX."in_BU_6-7".DigitalInput05;
	Cyclic#1.BU[7].typIN.bElevatorDown AT %IX."in_BU_6-7".DigitalInput06;
	Cyclic#1.BU[6].typIN.bTestUnit AT %IX."in_BU_6-7".DigitalInput07;
	Cyclic#1.BU[7].typIN.bTestUnit AT %IX."in_BU_6-7".DigitalInput08;
	Cyclic#3.BU[6].typIN.bOnline AT %IX."in_BU_0-1".ModuleOk;
	Cyclic#3.BU[6].typOUT.bOnline AT %IX."out_BU_0-1".ModuleOk;
	Cyclic#1.BU[6].typOUT.bElevator AT %QX."out_BU_6-7".DigitalOutput01;
	Cyclic#1.BU[7].typOUT.bElevator AT %QX."out_BU_6-7".DigitalOutput02;
	Cyclic#1.BU[6].typOUT.bReleaseGripper AT %QX."out_BU_6-7".DigitalOutput03;
	Cyclic#1.BU[7].typOUT.bReleaseGripper AT %QX."out_BU_6-7".DigitalOutput04;
	Cyclic#3.BU[6].typOUT.bStopServo AT %QX."out_BU_6-7".DigitalOutput05;
	Cyclic#3.BU[7].typOUT.bStopServo AT %QX."out_BU_6-7".DigitalOutput06;
	Cyclic#3.BU[6].typOUT.bEndStageServo AT %QX."out_BU_6-7".DigitalOutput07;
	Cyclic#3.BU[7].typOUT.bEndStageServo AT %QX."out_BU_6-7".DigitalOutput08;
	Cyclic#3.BU[6].typOUT.bEnableServo AT %QX."out_BU_6-7".DigitalOutput09;
	Cyclic#3.BU[7].typOUT.bEnableServo AT %QX."out_BU_6-7".DigitalOutput10;
	Cyclic#1.BU[6].bAddFlower AT %QX."out_BU_6-7".DigitalOutput11; (*24 VDC / 0.5 A, source (test add active)*)
	Cyclic#1.BU[7].bAddFlower AT %QX."out_BU_6-7".DigitalOutput12; (*24 VDC / 0.5 A, source (Test add active)*)
	Cyclic#1.BU[8].typIN.bElevatorUp AT %IX."in_BU_8-9".DigitalInput01;
	Cyclic#1.BU[9].typIN.bElevatorUp AT %IX."in_BU_8-9".DigitalInput02;
	Cyclic#1.BU[8].typIN.bElevatorMid AT %IX."in_BU_8-9".DigitalInput03;
	Cyclic#1.BU[9].typIN.bElevatorMid AT %IX."in_BU_8-9".DigitalInput04;
	Cyclic#1.BU[8].typIN.bElevatorDown AT %IX."in_BU_8-9".DigitalInput05;
	Cyclic#1.BU[9].typIN.bElevatorDown AT %IX."in_BU_8-9".DigitalInput06;
	Cyclic#1.BU[8].typIN.bTestUnit AT %IX."in_BU_8-9".DigitalInput07;
	Cyclic#1.BU[9].typIN.bTestUnit AT %IX."in_BU_8-9".DigitalInput08;
	Cyclic#3.BU[8].typIN.bOnline AT %IX."in_BU_0-1".ModuleOk;
	Cyclic#3.BU[8].typOUT.bOnline AT %IX."out_BU_0-1".ModuleOk;
	Cyclic#1.BU[8].typOUT.bElevator AT %QX."out_BU_8-9".DigitalOutput01;
	Cyclic#1.BU[9].typOUT.bElevator AT %QX."out_BU_8-9".DigitalOutput02;
	Cyclic#1.BU[8].typOUT.bReleaseGripper AT %QX."out_BU_8-9".DigitalOutput03;
	Cyclic#1.BU[9].typOUT.bReleaseGripper AT %QX."out_BU_8-9".DigitalOutput04;
	Cyclic#3.BU[8].typOUT.bStopServo AT %QX."out_BU_8-9".DigitalOutput05;
	Cyclic#3.BU[9].typOUT.bStopServo AT %QX."out_BU_8-9".DigitalOutput06;
	Cyclic#3.BU[8].typOUT.bEndStageServo AT %QX."out_BU_8-9".DigitalOutput07;
	Cyclic#3.BU[9].typOUT.bEndStageServo AT %QX."out_BU_8-9".DigitalOutput08;
	Cyclic#3.BU[8].typOUT.bEnableServo AT %QX."out_BU_8-9".DigitalOutput09;
	Cyclic#3.BU[9].typOUT.bEnableServo AT %QX."out_BU_8-9".DigitalOutput10;
	Cyclic#1.BU[8].bAddFlower AT %QX."out_BU_8-9".DigitalOutput11; (*24 VDC / 0.5 A, source (test add active)*)
	Cyclic#1.BU[9].bAddFlower AT %QX."out_BU_8-9".DigitalOutput12; (*24 VDC / 0.5 A, source (Test add active)*)
	Cyclic#3.MBU.in_bElastiekOp1 AT %IX."in_MBU".DigitalInput01;
	Cyclic#3.MBU.in_bElastiekOp2 AT %IX."in_MBU".DigitalInput02;
	MCU.typIN.bEncPuls2 AT %IX."in_MBU".DigitalInput03;
	MBU.out_bBinder1 AT %QX."out_MBU".DigitalOutput01;
	MBU.out_bBinder2 AT %QX."out_MBU".DigitalOutput02;
	Cyclic#3.BU[0].typBunchBelts.packed.ModuleOk AT %IX."BuMotor1".ModuleOk;
	Cyclic#3.BU[0].typBunchBelts.packed.LCR AT %IW."BuMotor1".2002sub05_TPDO06_LCR_Motor_current_0_1_A;
	Cyclic#3.BU[0].typBunchBelts.packed.ETAD AT %IW."BuMotor1".6041sub00_TPDO01_ETAD_Status_word;
	Cyclic#3.BU[0].typBunchBelts.packed.ERRD AT %IW."BuMotor1".2029sub16_TPDO06_LFT_Last_detected_fault;
	Cyclic#3.BU[0].typBunchBelts.packed.CMDD AT %QW."BuMotor1".6040sub00_RPDO01_CMDD_Control_word;
	Cyclic#3.BU[0].typBunchBelts.packed.LFR AT %QW."BuMotor1".6042sub00_RPDO06_LFRD_Speed_setpoint_rpm;
	Cyclic#3.BU[0].typServo.bOnLine AT %IX."ServoUnit1".ModuleOk;
	Cyclic#3.BU[0].typServo.packed.CCON AT %QB."ServoUnit1".3000sub00_RPDO01_CCON;
	Cyclic#3.BU[0].typServo.packed.CPOS AT %QB."ServoUnit1".3001sub00_RPDO01_CPOS;
	Cyclic#3.BU[0].typServo.packed.PARA1 AT %QB."ServoUnit1".3003sub00_RPDO01_RES_DEM_VAL1_PARA1;
	Cyclic#3.BU[0].typServo.packed.PARA2 AT %QD."ServoUnit1".3004sub00_RPDO01_RES_DEM_VAL2_PARA2;
	Cyclic#3.BU[0].typServo.packed.SCON AT %IB."ServoUnit1".3020sub00_TPDO01_SCON;
	Cyclic#3.BU[0].typServo.packed.SPOS AT %IB."ServoUnit1".3021sub00_TPDO01_SPOS;
	Cyclic#3.BU[0].typServo.packed.VAL1 AT %IB."ServoUnit1".3023sub00_TPDO01_RSB_ACT_VAL1_SUCC_CNT;
	Cyclic#3.BU[0].typServo.packed.VAL2 AT %ID."ServoUnit1".3024sub00_TPDO01_ACT_POS_ACT_VAL2_ACT_POS;
	Cyclic#3.BU[1].typBunchBelts.packed.ModuleOk AT %IX."BuMotor2".ModuleOk;
	Cyclic#3.BU[1].typBunchBelts.packed.LCR AT %IW."BuMotor2".2002sub05_TPDO06_LCR_Motor_current_0_1_A;
	Cyclic#3.BU[1].typBunchBelts.packed.ETAD AT %IW."BuMotor2".6041sub00_TPDO01_ETAD_Status_word;
	Cyclic#3.BU[1].typBunchBelts.packed.ERRD AT %IW."BuMotor2".2029sub16_TPDO06_LFT_Last_detected_fault;
	Cyclic#3.BU[1].typBunchBelts.packed.CMDD AT %QW."BuMotor2".6040sub00_RPDO01_CMDD_Control_word;
	Cyclic#3.BU[1].typBunchBelts.packed.LFR AT %QW."BuMotor2".6042sub00_RPDO06_LFRD_Speed_setpoint_rpm;
	Cyclic#3.BU[1].typServo.bOnLine AT %IX."ServoUnit2".ModuleOk;
	Cyclic#3.BU[1].typServo.packed.CCON AT %QB."ServoUnit2".3000sub00_RPDO01_CCON;
	Cyclic#3.BU[1].typServo.packed.CPOS AT %QB."ServoUnit2".3001sub00_RPDO01_CPOS;
	Cyclic#3.BU[1].typServo.packed.PARA1 AT %QB."ServoUnit2".3003sub00_RPDO01_RES_DEM_VAL1_PARA1;
	Cyclic#3.BU[1].typServo.packed.PARA2 AT %QD."ServoUnit2".3004sub00_RPDO01_RES_DEM_VAL2_PARA2;
	Cyclic#3.BU[1].typServo.packed.SCON AT %IB."ServoUnit2".3020sub00_TPDO01_SCON;
	Cyclic#3.BU[1].typServo.packed.SPOS AT %IB."ServoUnit2".3021sub00_TPDO01_SPOS;
	Cyclic#3.BU[1].typServo.packed.VAL1 AT %IB."ServoUnit2".3023sub00_TPDO01_RSB_ACT_VAL1_SUCC_CNT;
	Cyclic#3.BU[1].typServo.packed.VAL2 AT %ID."ServoUnit2".3024sub00_TPDO01_ACT_POS_ACT_VAL2_ACT_POS;
	Cyclic#3.BU[2].typBunchBelts.packed.ModuleOk AT %IX."BuMotor3".ModuleOk;
	Cyclic#3.BU[2].typBunchBelts.packed.LCR AT %IW."BuMotor3".2002sub05_TPDO06_LCR_Motor_current_0_1_A;
	Cyclic#3.BU[2].typBunchBelts.packed.ETAD AT %IW."BuMotor3".6041sub00_TPDO01_ETAD_Status_word;
	Cyclic#3.BU[2].typBunchBelts.packed.ERRD AT %IW."BuMotor3".2029sub16_TPDO06_LFT_Last_detected_fault;
	Cyclic#3.BU[2].typBunchBelts.packed.CMDD AT %QW."BuMotor3".6040sub00_RPDO01_CMDD_Control_word;
	Cyclic#3.BU[2].typBunchBelts.packed.LFR AT %QW."BuMotor3".6042sub00_RPDO06_LFRD_Speed_setpoint_rpm;
	Cyclic#3.BU[2].typServo.bOnLine AT %IX."ServoUnit3".ModuleOk;
	Cyclic#3.BU[2].typServo.packed.CCON AT %QB."ServoUnit3".3000sub00_RPDO01_CCON;
	Cyclic#3.BU[2].typServo.packed.CPOS AT %QB."ServoUnit3".3001sub00_RPDO01_CPOS;
	Cyclic#3.BU[2].typServo.packed.PARA1 AT %QB."ServoUnit3".3003sub00_RPDO01_RES_DEM_VAL1_PARA1;
	Cyclic#3.BU[2].typServo.packed.PARA2 AT %QD."ServoUnit3".3004sub00_RPDO01_RES_DEM_VAL2_PARA2;
	Cyclic#3.BU[2].typServo.packed.SCON AT %IB."ServoUnit3".3020sub00_TPDO01_SCON;
	Cyclic#3.BU[2].typServo.packed.SPOS AT %IB."ServoUnit3".3021sub00_TPDO01_SPOS;
	Cyclic#3.BU[2].typServo.packed.VAL1 AT %IB."ServoUnit3".3023sub00_TPDO01_RSB_ACT_VAL1_SUCC_CNT;
	Cyclic#3.BU[2].typServo.packed.VAL2 AT %ID."ServoUnit3".3024sub00_TPDO01_ACT_POS_ACT_VAL2_ACT_POS;
	Cyclic#3.BU[3].typBunchBelts.packed.ModuleOk AT %IX."BuMotor4".ModuleOk;
	Cyclic#3.BU[3].typBunchBelts.packed.LCR AT %IW."BuMotor4".2002sub05_TPDO06_LCR_Motor_current_0_1_A;
	Cyclic#3.BU[3].typBunchBelts.packed.ETAD AT %IW."BuMotor4".6041sub00_TPDO01_ETAD_Status_word;
	Cyclic#3.BU[3].typBunchBelts.packed.ERRD AT %IW."BuMotor4".2029sub16_TPDO06_LFT_Last_detected_fault;
	Cyclic#3.BU[3].typBunchBelts.packed.CMDD AT %QW."BuMotor4".6040sub00_RPDO01_CMDD_Control_word;
	Cyclic#3.BU[3].typBunchBelts.packed.LFR AT %QW."BuMotor4".6042sub00_RPDO06_LFRD_Speed_setpoint_rpm;
	Cyclic#3.BU[3].typServo.bOnLine AT %IX."ServoUnit4".ModuleOk;
	Cyclic#3.BU[3].typServo.packed.CCON AT %QB."ServoUnit4".3000sub00_RPDO01_CCON;
	Cyclic#3.BU[3].typServo.packed.CPOS AT %QB."ServoUnit4".3001sub00_RPDO01_CPOS;
	Cyclic#3.BU[3].typServo.packed.PARA1 AT %QB."ServoUnit4".3003sub00_RPDO01_RES_DEM_VAL1_PARA1;
	Cyclic#3.BU[3].typServo.packed.PARA2 AT %QD."ServoUnit4".3004sub00_RPDO01_RES_DEM_VAL2_PARA2;
	Cyclic#3.BU[3].typServo.packed.SCON AT %IB."ServoUnit4".3020sub00_TPDO01_SCON;
	Cyclic#3.BU[3].typServo.packed.SPOS AT %IB."ServoUnit4".3021sub00_TPDO01_SPOS;
	Cyclic#3.BU[3].typServo.packed.VAL1 AT %IB."ServoUnit4".3023sub00_TPDO01_RSB_ACT_VAL1_SUCC_CNT;
	Cyclic#3.BU[3].typServo.packed.VAL2 AT %ID."ServoUnit4".3024sub00_TPDO01_ACT_POS_ACT_VAL2_ACT_POS;
	Cyclic#3.BU[4].typBunchBelts.packed.ModuleOk AT %IX."BuMotor5".ModuleOk;
	Cyclic#3.BU[4].typBunchBelts.packed.LCR AT %IW."BuMotor5".2002sub05_TPDO06_LCR_Motor_current_0_1_A;
	Cyclic#3.BU[4].typBunchBelts.packed.ETAD AT %IW."BuMotor5".6041sub00_TPDO01_ETAD_Status_word;
	Cyclic#3.BU[4].typBunchBelts.packed.ERRD AT %IW."BuMotor5".2029sub16_TPDO06_LFT_Last_detected_fault;
	Cyclic#3.BU[4].typBunchBelts.packed.CMDD AT %QW."BuMotor5".6040sub00_RPDO01_CMDD_Control_word;
	Cyclic#3.BU[4].typBunchBelts.packed.LFR AT %QW."BuMotor5".6042sub00_RPDO06_LFRD_Speed_setpoint_rpm;
	Cyclic#3.BU[4].typServo.bOnLine AT %IX."ServoUnit5".ModuleOk;
	Cyclic#3.BU[4].typServo.packed.CCON AT %QB."ServoUnit5".3000sub00_RPDO01_CCON;
	Cyclic#3.BU[4].typServo.packed.CPOS AT %QB."ServoUnit5".3001sub00_RPDO01_CPOS;
	Cyclic#3.BU[4].typServo.packed.PARA1 AT %QB."ServoUnit5".3003sub00_RPDO01_RES_DEM_VAL1_PARA1;
	Cyclic#3.BU[4].typServo.packed.PARA2 AT %QD."ServoUnit5".3004sub00_RPDO01_RES_DEM_VAL2_PARA2;
	Cyclic#3.BU[4].typServo.packed.SCON AT %IB."ServoUnit5".3020sub00_TPDO01_SCON;
	Cyclic#3.BU[4].typServo.packed.SPOS AT %IB."ServoUnit5".3021sub00_TPDO01_SPOS;
	Cyclic#3.BU[4].typServo.packed.VAL1 AT %IB."ServoUnit5".3023sub00_TPDO01_RSB_ACT_VAL1_SUCC_CNT;
	Cyclic#3.BU[4].typServo.packed.VAL2 AT %ID."ServoUnit5".3024sub00_TPDO01_ACT_POS_ACT_VAL2_ACT_POS;
	Cyclic#3.BU[5].typBunchBelts.packed.ModuleOk AT %IX."BuMotor6".ModuleOk;
	Cyclic#3.BU[5].typBunchBelts.packed.LCR AT %IW."BuMotor6".2002sub05_TPDO06_LCR_Motor_current_0_1_A;
	Cyclic#3.BU[5].typBunchBelts.packed.ETAD AT %IW."BuMotor6".6041sub00_TPDO01_ETAD_Status_word;
	Cyclic#3.BU[5].typBunchBelts.packed.ERRD AT %IW."BuMotor6".2029sub16_TPDO06_LFT_Last_detected_fault;
	Cyclic#3.BU[5].typBunchBelts.packed.CMDD AT %QW."BuMotor6".6040sub00_RPDO01_CMDD_Control_word;
	Cyclic#3.BU[5].typBunchBelts.packed.LFR AT %QW."BuMotor6".6042sub00_RPDO06_LFRD_Speed_setpoint_rpm;
	Cyclic#3.BU[5].typServo.bOnLine AT %IX."ServoUnit6".ModuleOk;
	Cyclic#3.BU[5].typServo.packed.CCON AT %QB."ServoUnit6".3000sub00_RPDO01_CCON;
	Cyclic#3.BU[5].typServo.packed.CPOS AT %QB."ServoUnit6".3001sub00_RPDO01_CPOS;
	Cyclic#3.BU[5].typServo.packed.PARA1 AT %QB."ServoUnit6".3003sub00_RPDO01_RES_DEM_VAL1_PARA1;
	Cyclic#3.BU[5].typServo.packed.PARA2 AT %QD."ServoUnit6".3004sub00_RPDO01_RES_DEM_VAL2_PARA2;
	Cyclic#3.BU[5].typServo.packed.SCON AT %IB."ServoUnit6".3020sub00_TPDO01_SCON;
	Cyclic#3.BU[5].typServo.packed.SPOS AT %IB."ServoUnit6".3021sub00_TPDO01_SPOS;
	Cyclic#3.BU[5].typServo.packed.VAL1 AT %IB."ServoUnit6".3023sub00_TPDO01_RSB_ACT_VAL1_SUCC_CNT;
	Cyclic#3.BU[5].typServo.packed.VAL2 AT %ID."ServoUnit6".3024sub00_TPDO01_ACT_POS_ACT_VAL2_ACT_POS;
	Cyclic#3.BU[6].typBunchBelts.packed.ModuleOk AT %IX."BuMotor7".ModuleOk;
	Cyclic#3.BU[6].typBunchBelts.packed.LCR AT %IW."BuMotor7".2002sub05_TPDO06_LCR_Motor_current_0_1_A;
	Cyclic#3.BU[6].typBunchBelts.packed.ETAD AT %IW."BuMotor7".6041sub00_TPDO01_ETAD_Status_word;
	Cyclic#3.BU[6].typBunchBelts.packed.ERRD AT %IW."BuMotor7".2029sub16_TPDO06_LFT_Last_detected_fault;
	Cyclic#3.BU[6].typBunchBelts.packed.CMDD AT %QW."BuMotor7".6040sub00_RPDO01_CMDD_Control_word;
	Cyclic#3.BU[6].typBunchBelts.packed.LFR AT %QW."BuMotor7".6042sub00_RPDO06_LFRD_Speed_setpoint_rpm;
	Cyclic#3.BU[6].typServo.bOnLine AT %IX."ServoUnit7".ModuleOk;
	Cyclic#3.BU[6].typServo.packed.CCON AT %QB."ServoUnit7".3000sub00_RPDO01_CCON;
	Cyclic#3.BU[6].typServo.packed.CPOS AT %QB."ServoUnit7".3001sub00_RPDO01_CPOS;
	Cyclic#3.BU[6].typServo.packed.PARA1 AT %QB."ServoUnit7".3003sub00_RPDO01_RES_DEM_VAL1_PARA1;
	Cyclic#3.BU[6].typServo.packed.PARA2 AT %QD."ServoUnit7".3004sub00_RPDO01_RES_DEM_VAL2_PARA2;
	Cyclic#3.BU[6].typServo.packed.SCON AT %IB."ServoUnit7".3020sub00_TPDO01_SCON;
	Cyclic#3.BU[6].typServo.packed.SPOS AT %IB."ServoUnit7".3021sub00_TPDO01_SPOS;
	Cyclic#3.BU[6].typServo.packed.VAL1 AT %IB."ServoUnit7".3023sub00_TPDO01_RSB_ACT_VAL1_SUCC_CNT;
	Cyclic#3.BU[6].typServo.packed.VAL2 AT %ID."ServoUnit7".3024sub00_TPDO01_ACT_POS_ACT_VAL2_ACT_POS;
	Cyclic#3.BU[7].typBunchBelts.packed.ModuleOk AT %IX."BuMotor8".ModuleOk;
	Cyclic#3.BU[7].typBunchBelts.packed.LCR AT %IW."BuMotor8".2002sub05_TPDO06_LCR_Motor_current_0_1_A;
	Cyclic#3.BU[7].typBunchBelts.packed.ETAD AT %IW."BuMotor8".6041sub00_TPDO01_ETAD_Status_word;
	Cyclic#3.BU[7].typBunchBelts.packed.ERRD AT %IW."BuMotor8".2029sub16_TPDO06_LFT_Last_detected_fault;
	Cyclic#3.BU[7].typBunchBelts.packed.CMDD AT %QW."BuMotor8".6040sub00_RPDO01_CMDD_Control_word;
	Cyclic#3.BU[7].typBunchBelts.packed.LFR AT %QW."BuMotor8".6042sub00_RPDO06_LFRD_Speed_setpoint_rpm;
	Cyclic#3.BU[7].typServo.bOnLine AT %IX."ServoUnit8".ModuleOk;
	Cyclic#3.BU[7].typServo.packed.CCON AT %QB."ServoUnit8".3000sub00_RPDO01_CCON;
	Cyclic#3.BU[7].typServo.packed.CPOS AT %QB."ServoUnit8".3001sub00_RPDO01_CPOS;
	Cyclic#3.BU[7].typServo.packed.PARA1 AT %QB."ServoUnit8".3003sub00_RPDO01_RES_DEM_VAL1_PARA1;
	Cyclic#3.BU[7].typServo.packed.PARA2 AT %QD."ServoUnit8".3004sub00_RPDO01_RES_DEM_VAL2_PARA2;
	Cyclic#3.BU[7].typServo.packed.SCON AT %IB."ServoUnit8".3020sub00_TPDO01_SCON;
	Cyclic#3.BU[7].typServo.packed.SPOS AT %IB."ServoUnit8".3021sub00_TPDO01_SPOS;
	Cyclic#3.BU[7].typServo.packed.VAL1 AT %IB."ServoUnit8".3023sub00_TPDO01_RSB_ACT_VAL1_SUCC_CNT;
	Cyclic#3.BU[7].typServo.packed.VAL2 AT %ID."ServoUnit8".3024sub00_TPDO01_ACT_POS_ACT_VAL2_ACT_POS;
	Cyclic#3.BU[8].typBunchBelts.packed.ModuleOk AT %IX."BuMotor9".ModuleOk;
	Cyclic#3.BU[8].typBunchBelts.packed.LCR AT %IW."BuMotor9".2002sub05_TPDO06_LCR_Motor_current_0_1_A;
	Cyclic#3.BU[8].typBunchBelts.packed.ETAD AT %IW."BuMotor9".6041sub00_TPDO01_ETAD_Status_word;
	Cyclic#3.BU[8].typBunchBelts.packed.ERRD AT %IW."BuMotor9".2029sub16_TPDO06_LFT_Last_detected_fault;
	Cyclic#3.BU[8].typBunchBelts.packed.CMDD AT %QW."BuMotor9".6040sub00_RPDO01_CMDD_Control_word;
	Cyclic#3.BU[8].typBunchBelts.packed.LFR AT %QW."BuMotor9".6042sub00_RPDO06_LFRD_Speed_setpoint_rpm;
	Cyclic#3.BU[8].typServo.bOnLine AT %IX."ServoUnit9".ModuleOk;
	Cyclic#3.BU[8].typServo.packed.CCON AT %QB."ServoUnit9".3000sub00_RPDO01_CCON;
	Cyclic#3.BU[8].typServo.packed.CPOS AT %QB."ServoUnit9".3001sub00_RPDO01_CPOS;
	Cyclic#3.BU[8].typServo.packed.PARA1 AT %QB."ServoUnit9".3003sub00_RPDO01_RES_DEM_VAL1_PARA1;
	Cyclic#3.BU[8].typServo.packed.PARA2 AT %QD."ServoUnit9".3004sub00_RPDO01_RES_DEM_VAL2_PARA2;
	Cyclic#3.BU[8].typServo.packed.SCON AT %IB."ServoUnit9".3020sub00_TPDO01_SCON;
	Cyclic#3.BU[8].typServo.packed.SPOS AT %IB."ServoUnit9".3021sub00_TPDO01_SPOS;
	Cyclic#3.BU[8].typServo.packed.VAL1 AT %IB."ServoUnit9".3023sub00_TPDO01_RSB_ACT_VAL1_SUCC_CNT;
	Cyclic#3.BU[8].typServo.packed.VAL2 AT %ID."ServoUnit9".3024sub00_TPDO01_ACT_POS_ACT_VAL2_ACT_POS;
	Cyclic#3.BU[9].typBunchBelts.packed.ModuleOk AT %IX."BuMotor10".ModuleOk;
	Cyclic#3.BU[9].typBunchBelts.packed.LCR AT %IW."BuMotor10".2002sub05_TPDO06_LCR_Motor_current_0_1_A;
	Cyclic#3.BU[9].typBunchBelts.packed.ETAD AT %IW."BuMotor10".6041sub00_TPDO01_ETAD_Status_word;
	Cyclic#3.BU[9].typBunchBelts.packed.ERRD AT %IW."BuMotor10".2029sub16_TPDO06_LFT_Last_detected_fault;
	Cyclic#3.BU[9].typBunchBelts.packed.CMDD AT %QW."BuMotor10".6040sub00_RPDO01_CMDD_Control_word;
	Cyclic#3.BU[9].typBunchBelts.packed.LFR AT %QW."BuMotor10".6042sub00_RPDO06_LFRD_Speed_setpoint_rpm;
	Cyclic#3.BU[9].typServo.bOnLine AT %IX."ServoUnit10".ModuleOk;
	Cyclic#3.BU[9].typServo.packed.CCON AT %QB."ServoUnit10".3000sub00_RPDO01_CCON;
	Cyclic#3.BU[9].typServo.packed.CPOS AT %QB."ServoUnit10".3001sub00_RPDO01_CPOS;
	Cyclic#3.BU[9].typServo.packed.PARA1 AT %QB."ServoUnit10".3003sub00_RPDO01_RES_DEM_VAL1_PARA1;
	Cyclic#3.BU[9].typServo.packed.PARA2 AT %QD."ServoUnit10".3004sub00_RPDO01_RES_DEM_VAL2_PARA2;
	Cyclic#3.BU[9].typServo.packed.SCON AT %IB."ServoUnit10".3020sub00_TPDO01_SCON;
	Cyclic#3.BU[9].typServo.packed.SPOS AT %IB."ServoUnit10".3021sub00_TPDO01_SPOS;
	Cyclic#3.BU[9].typServo.packed.VAL1 AT %IB."ServoUnit10".3023sub00_TPDO01_RSB_ACT_VAL1_SUCC_CNT;
	Cyclic#3.BU[9].typServo.packed.VAL2 AT %ID."ServoUnit10".3024sub00_TPDO01_ACT_POS_ACT_VAL2_ACT_POS;
	systemTime AT %ID."X20CP1585".SystemTime;
	systemTime AT %ID."X20CP1583".SystemTime;
	Cyclic#3.MCU.typChain.packed.ModuleOk AT %IX."ChainMotor".ModuleOk;
	Cyclic#3.MCU.typChain.packed.CMDD AT %QW."ChainMotor".6040sub00_RPDO01_CMDD_Control_word;
	Cyclic#3.MCU.typChain.packed.LFR AT %QW."ChainMotor".6042sub00_RPDO06_LFRD_Speed_setpoint_rpm;
	Cyclic#3.MCU.typChain.packed.ETAD AT %IW."ChainMotor".6041sub00_TPDO01_ETAD_Status_word;
	Cyclic#3.MCU.typChain.packed.LCR AT %IW."ChainMotor".2002sub05_TPDO06_LCR_Motor_current_0_1_A;
	Cyclic#3.MCU.typChain.packed.ERRD AT %IW."ChainMotor".2029sub16_TPDO06_LFT_Last_detected_fault;
	Cyclic#3.MBU.typKnifeUnit.packed.ModuleOk AT %IX."KnifeMotor".ModuleOk;
	Cyclic#3.MBU.typKnifeUnit.packed.CMDD AT %QW."KnifeMotor".6040sub00_RPDO01_CMDD_Control_word;
	Cyclic#3.MBU.typKnifeUnit.packed.LFR AT %QW."KnifeMotor".6042sub00_RPDO06_LFRD_Speed_setpoint_rpm;
	Cyclic#3.MBU.typKnifeUnit.packed.ETAD AT %IW."KnifeMotor".6041sub00_TPDO01_ETAD_Status_word;
	Cyclic#3.MBU.typKnifeUnit.packed.LCR AT %IW."KnifeMotor".2002sub05_TPDO06_LCR_Motor_current_0_1_A;
	Cyclic#3.MBU.typKnifeUnit.packed.ERRD AT %IW."KnifeMotor".2029sub16_TPDO06_LFT_Last_detected_fault;
	Cyclic#3.MBU.typBeltMotor1.packed.ModuleOk AT %IX."BeltMotor1".ModuleOk;
	Cyclic#2.MBU.typBeltMotor1.packed.CMDD AT %QW."BeltMotor1".6040sub00_RPDO01_CMDD_Control_word;
	Cyclic#3.MBU.typBeltMotor1.packed.LFR AT %QW."BeltMotor1".6042sub00_RPDO06_LFRD_Speed_setpoint_rpm;
	Cyclic#3.MBU.typBeltMotor1.packed.ETAD AT %IW."BeltMotor1".6041sub00_TPDO01_ETAD_Status_word;
	Cyclic#3.MBU.typBeltMotor1.packed.LCR AT %IW."BeltMotor1".2002sub05_TPDO06_LCR_Motor_current_0_1_A;
	Cyclic#3.MBU.typBeltMotor1.packed.ERRD AT %IW."BeltMotor1".2029sub16_TPDO06_LFT_Last_detected_fault;
	Cyclic#3.MBU.typBeltMotor2.packed.ModuleOk AT %IX."BeltMotor2".ModuleOk;
	Cyclic#3.MBU.typBeltMotor2.packed.CMDD AT %QW."BeltMotor2".6040sub00_RPDO01_CMDD_Control_word;
	Cyclic#3.MBU.typBeltMotor2.packed.LFR AT %QW."BeltMotor2".6042sub00_RPDO06_LFRD_Speed_setpoint_rpm;
	Cyclic#3.MBU.typBeltMotor2.packed.ETAD AT %IW."BeltMotor2".6041sub00_TPDO01_ETAD_Status_word;
	Cyclic#3.MBU.typBeltMotor2.packed.LCR AT %IW."BeltMotor2".2002sub05_TPDO06_LCR_Motor_current_0_1_A;
	Cyclic#3.MBU.typBeltMotor2.packed.ERRD AT %IW."BeltMotor2".2029sub16_TPDO06_LFT_Last_detected_fault;
	Cyclic#1.MCU.typOUT.bLightTrigger1 AT %QX."out_MCU_0".DigitalOutput02;
	can_diag:x20if1041map.comCOS AT %ID."X20IF1041_1".Communication_Change_of_State;
	can_diag:x20if1041map.comState AT %ID."X20IF1041_1".Communication_State;
	can_diag:x20if1041map.comError AT %ID."X20IF1041_1".Communication_Error;
	can_diag:x20if1041map.version AT %IW."X20IF1041_1".Version;
	can_diag:x20if1041map.watchdogTimeout AT %IW."X20IF1041_1".Watchdog_Timeout;
	can_diag:x20if1041map.watchdogHost AT %ID."X20IF1041_1".Host_Watchdog;
	can_diag:x20if1041map.errorCount AT %ID."X20IF1041_1".Error_Count;
	can_diag:x20if1041map.errorLogIndicator AT %ID."X20IF1041_1".Error_Log_Indicator;
	can_diag:x20if1041map.slaveState AT %ID."X20IF1041_1".Slave_State;
	can_diag:x20if1041map.slaveErrorLogIndicator AT %ID."X20IF1041_1".Slave_Error_Log_Indicator;
	can_diag:x20if1041map.slavesConfigured AT %ID."X20IF1041_1".Configured_Slaves;
	can_diag:x20if1041map.slavesActive AT %ID."X20IF1041_1".Active_Slaves;
	can_diag:x20if1041map.slavesFaulted AT %ID."X20IF1041_1".Faulted_Slaves;
END_VAR
```

## Configuration X20_85

CPU X20CP1583, AutomationRuntime V4.08, Build 4.1.2

### Task classes (Cpu.sw)
```
Cyclic#1 (cycle 10000 us, tolerance 10000 us):
  Shiftregis <- MainControlUnit.Shiftregister.prg  // Control for chain sensor
  Simulation <- MainControlUnit.Simulation.prg
  Main <- MainControlUnit.Main.prg
Cyclic#2 (cycle 20000 us, tolerance 20000 us):
  IOpolling <- IOHandling.IOpolling.prg
Cyclic#3 (cycle 50000 us, tolerance 50000 us):
  BU_1 <- BunchUnits.BU_1.prg
  SC_1 <- BunchUnits.SC_1.prg
  BeltContro <- MainBeltUnit.BeltControl.prg
  RS_I <- BunchUnits.RS_I.prg
  BU_2 <- BunchUnits.BU_2.prg
Cyclic#4 (cycle 100000 us, tolerance 100000 us):
  ErrorHandl <- Exceptionhandling.ErrorHandling.prg
  can_diag <- Exceptionhandling.can_diag.prg
  SC_2 <- BunchUnits.SC_2.prg
Cyclic#5 (cycle 200000 us, tolerance 200000 us):
  Init <- BunchUnits.Init.prg
  Sender <- Lichtkrant.Sender.prg
VcDataObjects: BU_Gui <- Visualisation.BU_Gui_Resized.dob [disabled], Mobile <- Visualisation.Mobile.dob
Binaries: vccnum, arialbd, vcdsloc, vcfntttf, vcdsint, vcshared, vcrt, vcbclass, vcfile, vccbtn, vcresman, vcalarm, vcpdsw, arial, vccovl, vcgclass, Mobile02, Mobile03, vccddbox, vccpopup, vccdt, vcctext, vccshape, vccbmp, vcctrend, BU_Gui02, BU_Gui03, vccslider, asnxdb1, arconfig, asfw, ashwd, iomap, sysconf, vcpfx20, vcpdvnc, BU_Gui01, vctcal, vcpkat, vcnet, vcmgr, vcchspot, vccbar, vcclbox, vcchtml, vccstr, vccline, vccscale, vccalarm, vccgauge, vccurl, vcxml, asnxdb2, OpcUaMap
Libraries: sys_lib, Runtime, astime, asieccon, AsTCP, brsystem, asstring, standard, PulsGen, AsNxCoM, Inverter, BULib, Servo, SDO, dvframe, Lichtkrant, Chain, AsBrStr, hex2dec, Serial, SensContr, MBU_lib, IecCheck, dataobj, fileio, AsArLog, ashw, Hardware
```

### Hardware
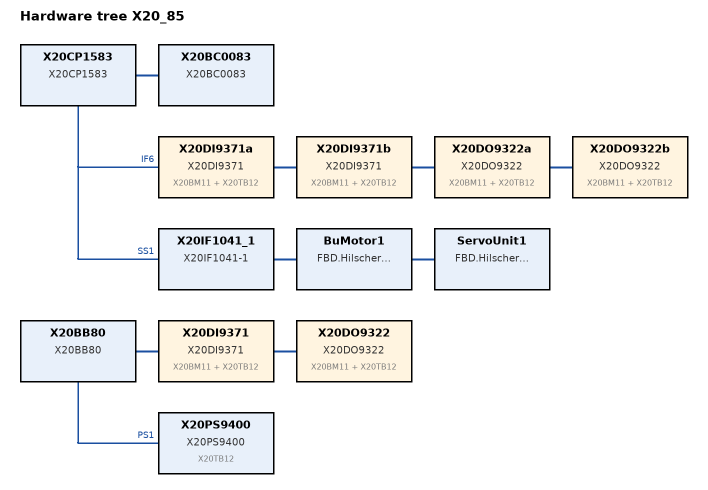
```
BuMotor1 : FBD.Hilscher.COGenSlaveDTM.ACOPOSinverter X64 (ACOPOSinverter_X64.eds) v0.0.0.0 (Disabled=true, OrderNumber=ACOPOSinverter_X64__ACOPOSinverter_X64_eds_)  [CAN1 -> X20IF1041_1.IF1 (NodeNumber=2)]
  DtmId = 520f109c-8a04-46dd-8e76-7a447e5455b3
  ChannelBlocks_4245d60c-4025-4738-9a65-21987dd3707d  // Receive PDO1 parameter
  IO_4f34897b-0599-4afc-bc07-33628c013aff  // 2 Byte(s)
  ChannelBlocks_0335e6f3-888f-4d7d-829a-9898c37542a9  // Receive PDO6 parameter
  IO_50b5ca40-4e68-4664-be22-8b76906fab27  // 2 Byte(s)
  IO_10550878-8dc2-41ba-811a-c05c81e89d01  // 2 Byte(s)
  IO_25fd8346-f4aa-4418-a5d6-7068a6b526e1  // 2 Byte(s)
  ChannelBlocks_7c414cbb-0829-4fd4-864b-4032604ecd8e  // Transmit PDO1 parameter
  IO_83b516ec-72a3-446e-8429-0ad1377fdfee  // 2 Byte(s)
  ChannelBlocks_9f9acb42-f5d2-4e8a-8344-f38ad1a7f190  // Transmit PDO6 parameter
  IO_92f15d74-1e81-46d7-829f-24ce734b661e  // 2 Byte(s)
  IO_d337187c-c96f-49e7-8373-6b2e635ca200  // 2 Byte(s)
  IO_2d8a46fa-e3de-4536-a3d0-b02273b535ea  // 2 Byte(s)
  IO_2687edec-612a-4449-9368-973e24b08730  // 2 Byte(s)
ServoUnit1 : FBD.Hilscher.COGenSlaveDTM.CMMS-ST (FHPP) (CMMS-ST_CAN_FHPP.eds) v0.0.0.0 (Disabled=true, OrderNumber=CMMS_ST__FHPP___CMMS_ST_CAN_FHPP_eds_)  [CAN1 -> BuMotor1.CAN2 (NodeNumber=3)]
  DtmId = 290e3f56-8804-408a-819e-215e2a6fc5b9
  ChannelBlocks_4f44d0a0-7e33-4b44-bcef-51cba8d2b404  // receive_pdo_parameter_RPDO1
  IO_dbcc41a7-80b1-4b69-beec-51c04bd492fa  // 1 Byte(s)
  IO_bf22bdb8-6ebe-49a8-9a86-d11de4076c69  // 1 Byte(s)
  IO_aa17c508-039e-415d-96d2-19732218c126  // 1 Byte(s)
  IO_09f76f3a-8376-4558-b0e0-92e3e64328f6  // 1 Byte(s)
  IO_a1aa309e-859d-47ed-b57a-60e340d58615  // 4 Byte(s)
  ChannelBlocks_5200326a-4d38-4545-b874-8c4e8a22abba  // receive_pdo_parameter_RPDO2
  IO_4bbe3f78-c0dd-4715-b158-ab57a88c820a  // 1 Byte(s)
  IO_88cea9be-7673-4fb7-b159-a4da5400030d  // 1 Byte(s)
  IO_fdb88a13-579a-46e1-bff0-5b689027fbbf  // 2 Byte(s)
  IO_6a651699-bb20-43ab-82e1-f3a21ac36695  // 4 Byte(s)
  ChannelBlocks_8f01dda6-605c-44a0-848e-8d91e3a01139  // transmit_pdo_parameter_TPDO1
  IO_86ef7406-0d00-4555-8673-a27d6f573e05  // 1 Byte(s)
  IO_429be286-32cc-47f6-9fd6-f9dcf4e5c9cd  // 1 Byte(s)
  IO_c044d5fb-d6d1-4e7e-bdb7-3600cdc77a40  // 1 Byte(s)
  IO_24252208-8ac1-48ed-9f4e-331b3da5bbab  // 1 Byte(s)
  IO_2c640d8e-bd0f-46a9-9b5c-535adbabdbf2  // 4 Byte(s)
  ChannelBlocks_760431be-4bac-4ae2-8acb-7bd365a52128  // transmit_pdo_parameter_TPDO2
  IO_6f64932a-a5d3-4116-971a-e159412b624e  // 1 Byte(s)
  IO_6efe3d3b-f204-43fd-99be-45c0a2d162e0  // 1 Byte(s)
  IO_97e982db-02f7-499d-997e-e363b64c2f11  // 2 Byte(s)
  IO_1d900de9-9c68-4dcb-9b35-1b1226599975  // 4 Byte(s)
X20BB80 : X20BB80 v1.0.0.2 (Disabled=true)
  Connector IF1 (Disabled=true)
    BusLength = 100
X20BC0083 : X20BC0083 v2.1.0.0 (Disabled=true)  [PLK1 -> X20CP1583.IF3 (NodeNumber=1); SL -> X20BB80.SL1]
X20BM11a : X20BM11 v1.0.0.0 (Disabled=true)  [X2X1 -> X20BB80.IF1]
X20BM11b : X20BM11 v1.0.0.0 (Disabled=true)  [X2X1 -> X20BM11a.X2X2]
X20BM11c : X20BM11 v1.0.0.0  [X2X1 -> X20BM11g.X2X2]
X20BM11e : X20BM11 v1.0.0.0  [X2X1 -> X20BM11c.X2X2]
X20BM11f : X20BM11 v1.0.0.0  [X2X1 -> X20CP1583.IF6]
X20BM11g : X20BM11 v1.0.0.0  [X2X1 -> X20BM11f.X2X2]
X20CP1583 : X20CP1583 v1.0.4.0
  Connector IF2:
    ActivateDevice = 1
    EthInterfaceRedundant = 0
    HostName = x1585
    Mode = DHCP Server
    InternetAddress = 10.0.1.156
    Lease1
    LeaseName1 = NOP
    LeaseStartAddress1 = 10.0.1.100
    LeaseStopAddress1 = 10.0.1.120
    LeaseTimeout1 = -1
    Vnc1
    VncVcObjectName1 = BU_Gui
    VncKeyMappingFile1 = VC\PS2-Keyboard.dis
    Vnc2
    VncVcObjectName2 = Mobile
    VncKeyMappingFile2 = VC\PS2-Keyboard1.dis
    VncPortNumber2 = 5901
  Connector IF3:
    EplInterfaceRedundant = 0
    EplEthInterfaceRedundant = 0
  Connector IF6:
    ActivateX2X = 0
  ConfigurationID = The_Magnifica_v0158_X20_85
  TimerDeviceType = SWIOTIMER
  Cyclic1Duration = 10000
  Cyclic1Tolerance = 10000
  Cyclic2Duration = 20000
  Cyclic2Tolerance = 20000
  Cyclic3Duration = 50000
  Cyclic3Tolerance = 50000
  Cyclic4Duration = 100000
  Cyclic4Tolerance = 100000
  Cyclic5Duration = 200000
  Cyclic5Tolerance = 200000
  Cyclic6Duration = 500000
  Cyclic6Tolerance = 500000
  Cyclic7Duration = 1000000
  Cyclic7Tolerance = 1000000
  Cyclic8Duration = 10000
  Cyclic8Tolerance = 30000000
  ActivateOpcUa = 1
  OpcUaAnonymous = 1
X20DI9371 : X20DI9371 v1.0.1.2 (Disabled=true)  [SS1 -> X20TB12b.SS; SL -> X20BM11a.SL1]
  Supervision = off
X20DI9371a : X20DI9371 v1.0.1.2  [SS1 -> X20TB12g.SS; SL -> X20BM11f.SL1]
  Supervision = off
X20DI9371b : X20DI9371 v1.0.1.2  [SS1 -> X20TB12h.SS; SL -> X20BM11g.SL1]
  Supervision = off
X20DO9322 : X20DO9322 v1.0.2.2 (Disabled=true)  [SS1 -> X20TB12c.SS; SL -> X20BM11b.SL1]
  Supervision = off
X20DO9322a : X20DO9322 v1.0.2.2  [SS1 -> X20TB12d.SS; SL -> X20BM11c.SL1]
  Supervision = off
X20DO9322b : X20DO9322 v1.0.2.2  [SS1 -> X20TB12f.SS; SL -> X20BM11e.SL1]
  Supervision = off
X20IF1041_1 : X20IF1041-1 v1.1.1.1 (Disabled=true)  [SS -> X20CP1583.SS1]
  Connector IF1 (Disabled=true)
    DtmRef = FBDIF.Hilscher.COMDtmNX.NETX 100 CO/COM
    DtmId = d03e33dc-0cc2-4952-a399-e832e4fc0471
  ConfigFile = X20IF1041_1.dtm
  ConfigModule = asnxdb1
X20PS9400 : X20PS9400 v1.0.2.1 (Disabled=true)  [SS1 -> X20TB12a.SS; PS -> X20BB80.PS1]
X20TB12a : X20TB12 v1.0.0.0 (Disabled=true)
X20TB12b : X20TB12 v1.0.0.0 (Disabled=true)
X20TB12c : X20TB12 v1.0.0.0 (Disabled=true)
X20TB12d : X20TB12 v1.0.0.0
X20TB12f : X20TB12 v1.0.0.0
X20TB12g : X20TB12 v1.0.0.0
X20TB12h : X20TB12 v1.0.0.0
```

### IoMap.iom - X20CP1583/IoMap.iom
```iecst
(********************************************************************
 * COPYRIGHT --
 ********************************************************************
 * File: IoMap.iom
 * Author: ronspa
 * Created: January 19, 2015
 ********************************************************************
 * IO mapping file
 ********************************************************************)
VAR_CONFIG
	BU[0].typeInterface.bReset AT %IX."X20DI9371".DigitalInput02;
	BU[0].typIN.bElevatorUp AT %IX."X20DI9371".DigitalInput03;
	BU[0].typIN.bElevatorMid AT %IX."X20DI9371".DigitalInput04;
	BU[0].typIN.bElevatorDown AT %IX."X20DI9371".DigitalInput05;
	in_bModule1[0] AT %IX."X20DI9371".DigitalInput06;
	in_bModule1[1] AT %IX."X20DI9371".DigitalInput07;
	in_bModule1[3] AT %IX."X20DI9371".DigitalInput09;
	in_bModule1[4] AT %IX."X20DI9371".DigitalInput10;
	in_bModule1[5] AT %IX."X20DI9371".DigitalInput11;
	in_bModule1[6] AT %IX."X20DI9371".DigitalInput12;
	in_bModule1[2] AT %IX."X20DI9371".DigitalInput08;
	BU[0].typOUT.bActivateGripper AT %QX."X20DO9322".DigitalOutput01;
	BU[0].typOUT.bBunchGripper AT %QX."X20DO9322".DigitalOutput02;
	BU[0].typOUT.bElevator AT %QX."X20DO9322".DigitalOutput03;
	BU[0].typOUT.bReleaseGripper AT %QX."X20DO9322".DigitalOutput04;
	BU[1].typOUT.bActivateGripper AT %QX."X20DO9322".DigitalOutput07;
	BU[1].typOUT.bBunchGripper AT %QX."X20DO9322".DigitalOutput08;
	BU[1].typOUT.bElevator AT %QX."X20DO9322".DigitalOutput09;
	BU[1].typOUT.bReleaseGripper AT %QX."X20DO9322".DigitalOutput10;
	MBU.out_bBinder1 AT %QX."X20DO9322".DigitalOutput11;
	MBU.out_bBinder2 AT %QX."X20DO9322".DigitalOutput12;
	out_bModule1[0] AT %QX."X20DO9322".DigitalOutput05;
	out_bModule1[1] AT %QX."X20DO9322".DigitalOutput06;
	MCU.typOUT.bCamTrigger1 AT %QX."X20DO9322a".DigitalOutput01;
	MCU.typOUT.bLightTrigger1 AT %QX."X20DO9322a".DigitalOutput02;
	MCU.typOUT.bCamTrigger2 AT %QX."X20DO9322a".DigitalOutput03;
	MCU.typOUT.bCamTrigger3 AT %QX."X20DO9322a".DigitalOutput05;
	MCU.typOUT.bCamTrigger4 AT %QX."X20DO9322a".DigitalOutput07;
	MCU.typOUT.bLightTrigger2 AT %QX."X20DO9322a".DigitalOutput04;
	MCU.typOUT.bLightTrigger3 AT %QX."X20DO9322a".DigitalOutput06;
	MCU.typOUT.bLightTrigger4 AT %QX."X20DO9322a".DigitalOutput08;
	BU[0].typBunchBelts.packed.LCR AT %IW."BuMotor1".2002sub05_TPDO06_LCR_Motor_current_0_1_A;
	BU[0].typBunchBelts.packed.CMDD AT %QW."BuMotor1".6040sub00_RPDO01_CMDD_Control_word;
	BU[0].typBunchBelts.packed.ETAD AT %IW."BuMotor1".6041sub00_TPDO01_ETAD_Status_word;
	BU[0].typBunchBelts.packed.LFR AT %QW."BuMotor1".6042sub00_RPDO06_LFRD_Speed_setpoint_rpm;
	BU[0].typBunchBelts.packed.ModuleOk AT %IX."BuMotor1".ModuleOk;
	BU[0].typBunchBelts.packed.ERRD AT %IW."BuMotor1".2029sub16_TPDO06_LFT_Last_detected_fault;
	BU[0].typServo.packed.CCON AT %QB."ServoUnit1".3000sub00_RPDO01_CCON;
	BU[0].typServo.packed.CPOS AT %QB."ServoUnit1".3001sub00_RPDO01_CPOS;
	BU[0].typServo.packed.PARA1 AT %QB."ServoUnit1".3003sub00_RPDO01_RES_DEM_VAL1_PARA1;
	BU[0].typServo.packed.PARA2 AT %QD."ServoUnit1".3004sub00_RPDO01_RES_DEM_VAL2_PARA2;
	BU[0].typServo.packed.SCON AT %IB."ServoUnit1".3020sub00_TPDO01_SCON;
	BU[0].typServo.packed.SPOS AT %IB."ServoUnit1".3021sub00_TPDO01_SPOS;
	BU[0].typServo.packed.VAL1 AT %IB."ServoUnit1".3023sub00_TPDO01_RSB_ACT_VAL1_SUCC_CNT;
	BU[0].typServo.packed.VAL2 AT %ID."ServoUnit1".3024sub00_TPDO01_ACT_POS_ACT_VAL2_ACT_POS;
	BU[0].typServo.bOnLine AT %IX."ServoUnit1".ModuleOk;
	Cyclic#1.systemTime AT %ID."X20CP1585".SystemTime;
	::systemTime AT %ID."X20CP1583".SystemTime;
END_VAR
```

## Logical view

Binary libraries used (declarations not repeated): Operator, Runtime, AsTime, AsIecCon, standard, sys_lib, AsTCP, brsystem, asstring, AsNxCoM, dvframe, AsBrStr, AsArLog

### Global.typ - Global data types
```iecst
(********************************************************************
 * COPYRIGHT --
 ********************************************************************
 * File: Global.typ
 * Author: jorkes
 * Created: July 07, 2014
 ********************************************************************
 * Global data types of project The_Magnifica
 ********************************************************************)

TYPE
	_visuInv : 	STRUCT
		bRunReverse : BOOL;
		bResetFault : BOOL;
		bRun : BOOL;
		bSetParams : BOOL;
		iSpeed : INT;
		bGetSpeed : BOOL;
		bSetSpeed : BOOL;
		bDriveReady : BOOL;
		bEnableManual : BOOL;
	END_STRUCT;
	enumError :
		(
		OK,
		EMERGENCYSTOP,
		DOOROPEN,
		AIRPRESSURE,
		BINDER,
		MOTORMALFUNCTION,
		SERVICEMODE,
		COMMUNICATION
		);
	enumState :
		( (*Machine State*)
		RUN,
		PAUZE, (*Not used*)
		STOP,
		EMPTY,
		SIMULATION
		);
	_muOUT : 	STRUCT
		bCamTrigger1 : BOOL := FALSE;
		bLightTrigger1 : BOOL := FALSE;
		bCamTrigger2 : BOOL := FALSE;
		bLightTrigger2 : BOOL := FALSE;
		bCamTrigger3 : BOOL := FALSE;
		bLightTrigger3 : BOOL := FALSE;
		bCamTrigger4 : BOOL := FALSE;
		bLightTrigger4 : BOOL := FALSE;
		bResetDoorOpen : BOOL := FALSE;
		bResetEmergencyStop : BOOL := FALSE;
		bGreenLight : BOOL := TRUE;
		bRedLight : BOOL := TRUE;
		bBuzzer : BOOL := FALSE;
		bMachineShutDown : BOOL := FALSE; (*Power down machine*)
	END_STRUCT;
	_muIN : 	STRUCT
		bEncPuls1 : BOOL := FALSE;
		bEncPuls2 : BOOL := FALSE;
		bDoorOpen : BOOL := FALSE;
		bEmergencyStop : BOOL := FALSE;
		bServiceMode : BOOL := FALSE;
		bBinder : BOOL := FALSE;
		bAirpressure : BOOL := FALSE;
		bJog : BOOL := FALSE;
	END_STRUCT;
	Register : 	STRUCT
		reg0 : INT;
		reg1 : INT;
		reg2 : INT;
		reg3 : INT;
		reg4 : INT;
		reg5 : INT;
		reg6 : INT;
		reg7 : INT;
		reg8 : INT;
		reg9 : INT;
		reg10 : INT;
		reg11 : INT;
		reg12 : INT;
		reg13 : INT;
		reg14 : INT;
		reg15 : INT;
		reg16 : INT;
		reg17 : INT;
		reg18 : INT;
		reg19 : INT;
	END_STRUCT;
	Trigger : 	STRUCT
		Coil0 : BOOL;
		Coil1 : BOOL;
		Coil2 : BOOL;
		Coil3 : BOOL;
		Coil4 : BOOL;
		Coil5 : BOOL;
		Coil6 : BOOL;
		Coil7 : BOOL;
		Coil8 : BOOL;
		Coil9 : BOOL;
	END_STRUCT;
	InterfaceMCU : 	STRUCT
		bEnabled : BOOL := FALSE; (*MCU Enabled*)
		bReset : BOOL := FALSE; (*MCU Reset *)
		bEmpty : BOOL := FALSE; (*MCU Empty machine*)
		bIsEmpty : BOOL := FALSE; (*Machine is empty*)
		bRun : BOOL := FALSE; (*MCU Start running*)
		bToggle : BOOL := FALSE; (*Toggle MCU (auto reset)*)
		bSimulation : BOOL := FALSE; (*Should be false on system*)
		bBuzzer : BOOL := FALSE; (*Buzzer by user*)
		bCamTrigManual : BOOL := FALSE; (*Manual camtrigger*)
		State : enumState := STOP;
		iJogSpeed : INT := 300; (*20Hz*)
		iNormalSpeed : INT := 1500; (*50Hz*)
		iRegisters : Register;
		bTriggers : Trigger;
		iBUEnabledMask : INT := 0;
	END_STRUCT;
	SettingsType : 	STRUCT  (*Settings worden overschreven vanuit de PC*)
		Mode : INT; (*0=STOP, 1=RUN, 2=EMPTY*)
		CamDelay1 : INT := 10; (*ms*)
		CamDelay2 : INT := 10; (*ms*)
		CamDelay3 : INT := 10; (*ms*)
		CamDelay4 : INT := 10; (*ms*)
		CamPosition1 : INT := 8; (*0-15*)
		CamPosition2 : INT := 12; (*0-15*)
		CamPosition3 : INT := 14; (*0-15*)
		CamPosition4 : INT := 6; (*0-15*)
		CamPulseLength : INT := 10; (*ms*)
		FlitsBefore : INT := 20; (*ms*)
		FlitsAfter : INT := 15; (*ms*)
		RejectPosition : INT := 151; (*Position relative to gripper *16*)
		BosUnit1Position : INT; (*Position relative to gripper *16*)
		BosUnit2Position : INT; (*Position relative to gripper *16*)
		BosUnit3Position : INT; (*Position relative to gripper *16*)
		BosUnit4Position : INT; (*Position relative to gripper *16*)
		BosUnit5Position : INT; (*Position relative to gripper *16*)
		BosUnit6Position : INT; (*Position relative to gripper *16*)
		BosUnit7Position : INT; (*Position relative to gripper *16*)
		BosUnit8Position : INT; (*Position relative to gripper *16*)
		BosUnit9Position : INT; (*Position relative to gripper *16*)
		BosUnit10Position : INT; (*Position relative to gripper *16*)
		BU_BunchBeltTime : INT := 1200; (*ms dat de belt draait*)
		BU_ActivateReleaseTime : INT := 600; (*ms dat de dropper is activated*)
		HeartBeatTime : INT := 5000; (*ms*)
		iBUIdealReceivePosition : INT := 400;
		iBUIdealReceivePositionGui : INT; (*Buffer om de GU update in op te slaan*)
	END_STRUCT;
	MainControlUnit : 	STRUCT  (*Verzameling parameters hoofdkast*)
		typOUT : _muOUT;
		typIN : _muIN;
		typInterface : InterfaceMCU; (*Interface*)
		typChain : AcpInverter_typ;
		motChain : ACPinverter;
	END_STRUCT;
END_TYPE
```

### Global.var
```iecst
(********************************************************************
 * COPYRIGHT --
 ********************************************************************
 * File: Global.var
 * Author: jorkes
 * Created: July 07, 2014
 ********************************************************************
 * Global variables of project The_Magnifica
 ********************************************************************)
VAR
	testEnableBU : BOOL;
	ErrorState : enumError := OK;
	bGblRun : BOOL := FALSE; (*Boolean die aangeeft of de machine in bedrijf is*)
	bGblSimulation : BOOL := FALSE; (*Boolean die aangeeft of de machine in simulation staat*)
	usBunchUnitIdx : USINT := 0;
END_VAR
(*IO declarations*)
VAR
	in_bModule1 : ARRAY[0..11] OF BOOL;
	out_bModule1 : ARRAY[0..11] OF BOOL;
END_VAR
VAR CONSTANT
	BUCount : USINT := 10; (*NrOff BosUnuts*)
	Pi : REAL := 3.14;
END_VAR
(*Type declarations*)
VAR
	SHFTREG : Shiftregister;
	RU : BunchUnit; (*Reject unit*)
	MBU : MainbeltUnit; (*Mainbelt Unit (Bosbandkast)*)
	BU : ARRAY[0..9] OF BunchUnit; (*Bosunit*)
	MCU : MainControlUnit; (*Main Control Unit (Hoofdkast)*)
	systemTime : DINT;
END_VAR
(*Settings data from PC leading*)
VAR RETAIN
	Settings : SettingsType := (Mode:=0);
END_VAR
```

### Package Logical/Libraries - Global libraries

### Library Logical/Libraries/IecCheck (IEC) - A library implementing IEC check functions
Depends on: sys_lib, AsBrStr

#### IecCheck.fun - Exported functions and function blocks
```iecst
(********************************************************************
 * COPYRIGHT --
 ********************************************************************
 * Library: IecCheck
 * File: IecCheck.fun
 * Author: ronspa
 * Created: January 13, 2015
 ********************************************************************
 * Functions and function blocks of library IecCheck
 ********************************************************************)

FUNCTION CheckDivSint : SINT (* Check divisor for SINT division *)
	VAR_INPUT
		divisor : SINT;
	END_VAR
END_FUNCTION

FUNCTION CheckDivUsint : USINT (* Check divisor for USINT division *)
	VAR_INPUT
		divisor : USINT;
	END_VAR
END_FUNCTION

FUNCTION CheckDivInt : INT (* Check divisor for INT division *)
	VAR_INPUT
		divisor : INT;
	END_VAR
END_FUNCTION

FUNCTION CheckDivUint : UINT (* Check divisor for UINT division *)
	VAR_INPUT
		divisor : UINT;
	END_VAR
END_FUNCTION

FUNCTION CheckDivDint : DINT (* Check divisor for DINT division *)
	VAR_INPUT
		divisor : DINT;
	END_VAR
END_FUNCTION

FUNCTION CheckDivUdint : UDINT (* Check divisor for UDINT division *)
	VAR_INPUT
		divisor : UDINT;
	END_VAR
END_FUNCTION

FUNCTION CheckDivReal : REAL (* Check divisor for REAL division *)
	VAR_INPUT
		divisor : REAL;
	END_VAR
END_FUNCTION

FUNCTION CheckDivLReal : LREAL (* Check divisor for LREAL division, not available for SG3 and SGC *)
	VAR_INPUT
		divisor : LREAL;
	END_VAR
END_FUNCTION

FUNCTION CheckBounds : DINT (* Check range for array access *)
	VAR_INPUT
		index : DINT;
		lower : DINT;
		upper : DINT;
	END_VAR
END_FUNCTION

FUNCTION CheckRange : DINT (* Check range for enumeration *)
	VAR_INPUT
		value : DINT;
		lower : DINT;
		upper : DINT;
	END_VAR
END_FUNCTION

FUNCTION CheckSignedSubrange : DINT (* Check range for subrange of signed data types *)
	VAR_INPUT
		value : DINT;
		lower : DINT;
		upper : DINT;
	END_VAR
END_FUNCTION

FUNCTION CheckUnsignedSubrange : UDINT (* Check range for subrange of unsigned data types *)
	VAR_INPUT
		value : UDINT;
		lower : UDINT;
		upper : UDINT;
	END_VAR
END_FUNCTION

FUNCTION CheckReadAccess : UDINT (* Check address when reading dynamic variables *)
	VAR_INPUT
		address : UDINT;
	END_VAR
END_FUNCTION

FUNCTION CheckWriteAccess : UDINT (* Check address when writing dynamic variables *)
	VAR_INPUT
		address : UDINT;
	END_VAR
END_FUNCTION

FUNCTION MakeEntry : UDINT (* Makes an entry (log book entry) in the error log book *)
	VAR
		taskname : STRING[30];
		group : USINT;
		status_name : UINT;
		out_text : STRING[80];
	END_VAR
	VAR_INPUT
		number : UINT;
		index : DINT;
		text : STRING[50];
	END_VAR
END_FUNCTION
```

#### IecCheck.st - Implementation file
```iecst
(********************************************************************
 * COPYRIGHT --
 ********************************************************************
 * Library: IecCheck
 * Author: ronspa
 * Created: January 13, 2015
 ********************************************************************
 * Implementation of library IecCheck
 ********************************************************************)

(* Check divisor for SINT division *)
FUNCTION CheckDivSint
	IF divisor=0 THEN
		CheckDivSint:=1;
		MakeEntry(55555,divisor,'CheckDivSint');
	ELSE
		CheckDivSint:=divisor;
	END_IF
END_FUNCTION

(* Check divisor for USINT division *)
FUNCTION CheckDivUsint
	IF divisor=0 THEN
		CheckDivUsint:=1;
		MakeEntry(55555,divisor,'CheckDivUsint');
	ELSE
		CheckDivUsint:=divisor;
	END_IF
END_FUNCTION

(* Check divisor for INT division *)
FUNCTION CheckDivInt
	IF divisor=0 THEN
		CheckDivInt:=1;
		MakeEntry(55555,divisor,'CheckDivInt');
	ELSE
		CheckDivInt:=divisor;
	END_IF
END_FUNCTION

(* Check divisor for UINT division *)
FUNCTION CheckDivUint
	IF divisor=0 THEN
		CheckDivUint:=1;
		MakeEntry(55555,divisor,'CheckDivUint');
	ELSE
		CheckDivUint:=divisor;
	END_IF
END_FUNCTION

(* Check divisor for DINT division *)
FUNCTION CheckDivDint
	IF divisor=0 THEN
		CheckDivDint:=1;
		MakeEntry(55555,divisor,'CheckDivDint');
	ELSE
		CheckDivDint:=divisor;
	END_IF
END_FUNCTION

(* Check divisor for UDINT division *)
FUNCTION CheckDivUdint
	IF divisor=0 THEN
		CheckDivUdint:=1;
		MakeEntry(55555,divisor,'CheckDivUdint');
	ELSE
		CheckDivUdint:=divisor;
	END_IF
END_FUNCTION

(* Check divisor for REAL division *)
FUNCTION CheckDivReal
	IF divisor=0 THEN
		CheckDivReal:=1;
		MakeEntry(55555,0,'CheckDivReal');
	ELSE
		CheckDivReal:=divisor;
	END_IF
END_FUNCTION

(* Check divisor for LREAL division *)
FUNCTION CheckDivLReal
	IF divisor=0 THEN
		CheckDivLReal:=1;
		MakeEntry(55555,0,'CheckDivLReal');
	ELSE
		CheckDivLReal:=divisor;
	END_IF
END_FUNCTION

(* Check range for array access *)
FUNCTION CheckBounds
	IF index < lower THEN
		CheckBounds := lower;
		MakeEntry(55555,index,'CheckBounds');
	ELSIF index > upper THEN
		CheckBounds := upper;
		MakeEntry(55555,index,'CheckBounds');
	ELSE
		CheckBounds := index;
	END_IF
	END_FUNCTION

(* Check range for enumeration *)
FUNCTION CheckRange
	IF value < lower THEN
		CheckRange := lower;
		MakeEntry(55555,value,'CheckRange');
	ELSIF value > upper THEN
		CheckRange := upper;
		MakeEntry(55555,value,'CheckRange');
	ELSE
		CheckRange := value;
	END_IF
END_FUNCTION

(* Check range for subrange of signed data types *)
FUNCTION CheckSignedSubrange
	IF value < lower THEN
		CheckSignedSubrange := lower;
		MakeEntry(55555,value,'CheckSignedSubrange');
	ELSIF value > upper THEN
		CheckSignedSubrange := upper;
		MakeEntry(55555,value,'CheckSignedSubrange');
	ELSE
		CheckSignedSubrange := value;
	END_IF
END_FUNCTION

(* Check range for subrange of unsigned data types *)
FUNCTION CheckUnsignedSubrange
	IF value < lower THEN
		CheckUnsignedSubrange := lower;
		MakeEntry(55555,value,'CheckUnsignedSubrange');
	ELSIF value > upper THEN
		CheckUnsignedSubrange := upper;
		MakeEntry(55555,value,'CheckUnsignedSubrange');
	ELSE
		CheckUnsignedSubrange := value;
	END_IF
END_FUNCTION

(* Check address when reading dynamic variables *)
FUNCTION CheckReadAccess
	IF address=0 THEN
		(* TODO: Insert an appropriate code, see AutomationStudio help for further information *)
		MakeEntry(55555,address,'Read from NULL');
	END_IF

	CheckReadAccess:=0;
END_FUNCTION

(* Check address when writing dynamic variables *)
FUNCTION CheckWriteAccess
	IF address=0 THEN
		(* TODO: Insert an appropriate code, see AutomationStudio help for further information *)
		MakeEntry(55555,address,'Write to NULL');
	END_IF

	CheckWriteAccess:=0;
END_FUNCTION

(* Makes an entry (log book entry) in the error log book *)
FUNCTION MakeEntry
		status_name := ST_name(0,ADR(taskname),ADR(group));

		brsstrcpy(ADR(out_text),ADR(text));
		brsstrcat(ADR(out_text),ADR(' > in task > '));
  		brsstrcat(ADR(out_text),ADR(taskname));
		MakeEntry := ADR(out_text);
		ERRxfatal(number,index,ADR(out_text));
END_FUNCTION
```

### Package Logical/MainControlUnit - Package

### Program Logical/MainControlUnit/Shiftregister (IEC) - Program
